KUKA KRL program: f1_Kuka_APT221T02S21.SRC

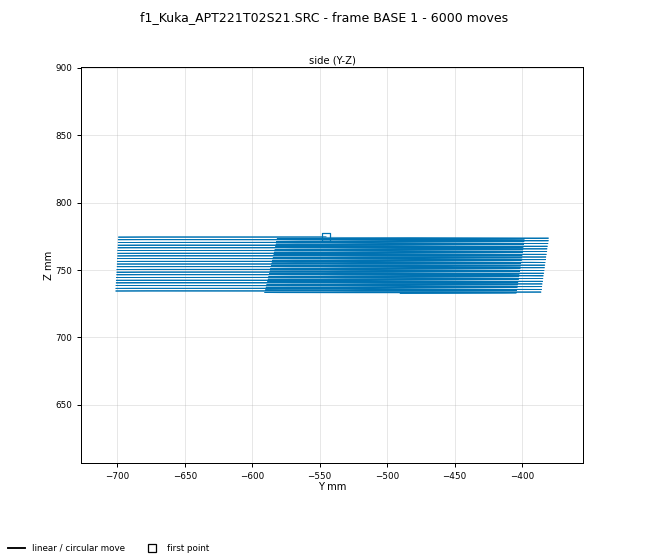
[picture p0: tool path of f1_Kuka_APT221T02S21.SRC in frame BASE 1, 6000 of 6001 moves have a stored position in this frame; points joined in program order, loops and branches not executed]
&ACCESS RVP
&REL 2
&PARAM TEMPLATE = C:\KRC\Roboter\Template\vorgabe
&PARAM EDITMASK = *
DEF f1_Kuka_APT221T02S21()


;FOLD INI;%{PE}%V3.2.0,%MKUKATPBASIS,%CINIT,%VCOMMON,%P
  ;FOLD BAS INI;%{E}%V3.2.0,%MKUKATPBASIS,%CINIT,%VINIT,%P
    GLOBAL INTERRUPT DECL 3 WHEN $STOPMESS==TRUE DO IR_STOPM ( )
    INTERRUPT ON 3
    BAS (#INITMOV,0 )
  ;ENDFOLD (BAS INI)
  ;FOLD USER INI;%{E}%V3.2.0,%MKUKATPUSER,%CINIT,%VINIT,%P
    ;Make your modifications here
  ;ENDFOLD (USER INI)
;ENDFOLD (INI)


;*** Make Null PTP Move
  PTP $pos_act

;*** Auto Load The Correct TOOL Data
  $tool=tool_data[2]

;*** Auto Load The Correct BASE Data
  $base=base_data[1]

  $ADVANCE = 5

;*** Restate Last Velocity
MMPM(30000.0)
SetRPM(8000)
LIN {X 0.178,Y -545.283,Z 774.689,A 0.000,B 0.000,C 90.000,E1 340.007} C_DIS
LIN {X 0.081,Y -552.448,Z 774.686,A 0.000,B 0.000,C 90.000,E1 339.464} C_DIS
LIN {X -0.341,Y -557.944,Z 774.683,A 0.000,B 0.000,C 90.000,E1 339.028} C_DIS
LIN {X 0.055,Y -564.478,Z 774.680,A 0.000,B 0.000,C 90.000,E1 338.358} C_DIS
LIN {X -0.146,Y -569.481,Z 774.677,A 0.000,B 0.000,C 90.000,E1 337.847} C_DIS
LIN {X -0.245,Y -575.503,Z 774.673,A 0.000,B 0.000,C 90.000,E1 337.177} C_DIS
LIN {X -0.071,Y -580.921,Z 774.669,A 0.000,B 0.000,C 90.000,E1 336.485} C_DIS
LIN {X 0.036,Y -588.085,Z 774.664,A 0.000,B 0.000,C 90.000,E1 335.537} C_DIS
LIN {X 0.195,Y -594.819,Z 774.659,A 0.000,B 0.000,C 90.000,E1 334.588} C_DIS
LIN {X -0.171,Y -602.961,Z 774.652,A 0.000,B 0.000,C 90.000,E1 333.435} C_DIS
LIN {X 0.164,Y -608.816,Z 774.647,A 0.000,B 0.000,C 90.000,E1 332.487} C_DIS
LIN {X 0.288,Y -616.060,Z 774.641,A 0.000,B 0.000,C 90.000,E1 331.307} C_DIS
LIN {X -0.314,Y -621.361,Z 774.636,A 0.000,B 0.000,C 90.000,E1 330.461} C_DIS
LIN {X -0.012,Y -626.573,Z 774.631,A 0.000,B 0.000,C 90.000,E1 329.537} C_DIS
LIN {X -0.196,Y -630.736,Z 774.627,A 0.000,B 0.000,C 90.000,E1 328.791} C_DIS
LIN {X 0.216,Y -635.263,Z 774.622,A 0.000,B 0.000,C 90.000,E1 327.867} C_DIS
LIN {X 0.137,Y -639.594,Z 774.617,A 0.000,B 0.000,C 90.000,E1 326.993} C_DIS
LIN {X -0.032,Y -644.812,Z 774.610,A 0.000,B 0.000,C 90.000,E1 325.881} C_DIS
LIN {X 0.321,Y -648.073,Z 774.606,A 0.000,B 0.000,C 90.000,E1 325.102} C_DIS
LIN {X 0.248,Y -652.167,Z 774.601,A 0.000,B 0.000,C 90.000,E1 324.116} C_DIS
LIN {X -0.231,Y -655.030,Z 774.597,A 0.000,B 0.000,C 90.000,E1 323.417} C_DIS
LIN {X -0.278,Y -659.576,Z 774.590,A 0.000,B 0.000,C 90.000,E1 322.190} C_DIS
LIN {X -0.255,Y -663.771,Z 774.583,A 0.000,B 0.000,C 90.000,E1 320.964} C_DIS
LIN {X -0.261,Y -667.644,Z 774.576,A 0.000,B 0.000,C 90.000,E1 319.747} C_DIS
LIN {X -0.199,Y -670.626,Z 774.571,A 0.000,B 0.000,C 90.000,E1 318.771} C_DIS
LIN {X -0.088,Y -674.036,Z 774.564,A 0.000,B 0.000,C 90.000,E1 317.553} C_DIS
LIN {X -0.395,Y -677.421,Z 774.556,A 0.000,B 0.000,C 90.000,E1 316.134} C_DIS
LIN {X -0.247,Y -679.532,Z 774.551,A 0.000,B 0.000,C 90.000,E1 315.162} C_DIS
LIN {X -0.071,Y -681.410,Z 774.546,A 0.000,B 0.000,C 90.000,E1 314.190} C_DIS
LIN {X -0.183,Y -684.457,Z 774.536,A 0.000,B 0.000,C 90.000,E1 312.528} C_DIS
LIN {X 0.094,Y -685.958,Z 774.531,A 0.000,B 0.000,C 90.000,E1 311.553} C_DIS
LIN {X -0.123,Y -687.339,Z 774.526,A 0.000,B 0.000,C 90.000,E1 310.620} C_DIS
LIN {X -0.184,Y -688.796,Z 774.519,A 0.000,B 0.000,C 90.000,E1 309.439} C_DIS
LIN {X -0.219,Y -690.150,Z 774.513,A 0.000,B 0.000,C 90.000,E1 308.257} C_DIS
LIN {X -0.241,Y -691.320,Z 774.506,A 0.000,B 0.000,C 90.000,E1 307.076} C_DIS
LIN {X -0.065,Y -692.595,Z 774.498,A 0.000,B 0.000,C 90.000,E1 305.644} C_DIS
LIN {X 0.083,Y -693.517,Z 774.492,A 0.000,B 0.000,C 90.000,E1 304.452} C_DIS
LIN {X -0.263,Y -694.752,Z 774.482,A 0.000,B 0.000,C 90.000,E1 302.832} C_DIS
LIN {X 0.389,Y -696.099,Z 774.473,A 0.000,B 0.000,C 90.000,E1 301.131} C_DIS
LIN {X -0.157,Y -696.863,Z 774.467,A 0.000,B 0.000,C 90.000,E1 300.001} C_DIS
LIN {X 0.174,Y -697.436,Z 774.459,A 0.000,B 0.000,C 90.000,E1 298.565} C_DIS
LIN {X 0.106,Y -698.271,Z 774.448,A 0.000,B 0.000,C 90.000,E1 296.693} C_DIS
LIN {X 0.045,Y -699.384,Z 774.438,A 0.000,B 0.000,C 90.000,E1 294.823} C_DIS
LIN {X 0.287,Y -699.299,Z 774.435,A 0.000,B 0.000,C 90.000,E1 294.335} C_DIS
LIN {X -0.084,Y -699.187,Z 774.434,A 0.000,B 0.000,C 90.000,E1 294.131} C_DIS
LIN {X 0.162,Y -697.937,Z 774.431,A 0.000,B 0.000,C 90.000,E1 293.643} C_DIS
LIN {X 0.423,Y -697.170,Z 774.430,A 0.000,B 0.000,C 90.000,E1 293.387} C_DIS
LIN {X -0.363,Y -696.496,Z 774.430,A 0.000,B 0.000,C 90.000,E1 293.334} C_DIS
LIN {X -0.234,Y -695.484,Z 774.429,A 0.000,B 0.000,C 90.000,E1 293.206} C_DIS
LIN {X 0.073,Y -690.561,Z 774.426,A 0.000,B 0.000,C 90.000,E1 292.717} C_DIS
LIN {X 0.260,Y -688.711,Z 774.426,A 0.000,B 0.000,C 90.000,E1 292.589} C_DIS
LIN {X -0.357,Y -684.254,Z 774.425,A 0.000,B 0.000,C 90.000,E1 292.461} C_DIS
LIN {X -0.332,Y -680.303,Z 774.424,A 0.000,B 0.000,C 90.000,E1 292.333} C_DIS
LIN {X -0.035,Y -674.173,Z 774.423,A 0.000,B 0.000,C 90.000,E1 292.153} C_DIS
LIN {X -0.204,Y -664.948,Z 774.422,A 0.000,B 0.000,C 90.000,E1 292.025} C_DIS
LIN {X 0.151,Y -654.378,Z 774.422,A 0.000,B 0.000,C 90.000,E1 291.844} C_DIS
LIN {X 0.228,Y -644.131,Z 774.421,A 0.000,B 0.000,C 90.000,E1 291.663} C_DIS
LIN {X -0.242,Y -627.380,Z 774.419,A 0.000,B 0.000,C 90.000,E1 291.354} C_DIS
LIN {X -0.025,Y -610.054,Z 774.416,A 0.000,B 0.000,C 90.000,E1 290.918} C_DIS
LIN {X 0.062,Y -589.210,Z 774.413,A 0.000,B 0.000,C 90.000,E1 290.355} C_DIS
LIN {X -0.059,Y -566.654,Z 774.409,A 0.000,B 0.000,C 90.000,E1 289.685} C_DIS
LIN {X 0.034,Y -560.006,Z 774.408,A 0.000,B 0.000,C 90.000,E1 289.396} C_DIS
LIN {X -0.146,Y -558.225,Z 774.407,A 0.000,B 0.000,C 90.000,E1 289.268} C_DIS
LIN {X 0.119,Y -557.105,Z 774.406,A 0.000,B 0.000,C 90.000,E1 289.141} C_DIS
LIN {X 0.082,Y -557.068,Z 774.406,A 0.000,B 0.000,C 90.000,E1 289.141} C_DIS
LIN {X 0.163,Y -555.965,Z 774.405,A 0.000,B 0.000,C 90.000,E1 288.852} C_DIS
LIN {X 0.333,Y -555.320,Z 774.403,A 0.000,B 0.000,C 90.000,E1 288.417} C_DIS
LIN {X -0.217,Y -554.804,Z 774.398,A 0.000,B 0.000,C 90.000,E1 287.638} C_DIS
LIN {X -0.240,Y -554.409,Z 774.393,A 0.000,B 0.000,C 90.000,E1 286.804} C_DIS
LIN {X 0.088,Y -553.379,Z 774.381,A 0.000,B 0.000,C 90.000,E1 284.537} C_DIS
LIN {X 0.284,Y -552.877,Z 774.373,A 0.000,B 0.000,C 90.000,E1 283.119} C_DIS
LIN {X -0.073,Y -552.310,Z 774.364,A 0.000,B 0.000,C 90.000,E1 281.478} C_DIS
LIN {X 0.115,Y -551.685,Z 774.353,A 0.000,B 0.000,C 90.000,E1 279.500} C_DIS
LIN {X 0.205,Y -551.129,Z 774.342,A 0.000,B 0.000,C 90.000,E1 277.530} C_DIS
LIN {X -0.087,Y -550.812,Z 774.337,A 0.000,B 0.000,C 90.000,E1 276.720} C_DIS
LIN {X 0.206,Y -550.219,Z 774.331,A 0.000,B 0.000,C 90.000,E1 275.568} C_DIS
LIN {X 0.119,Y -548.869,Z 774.320,A 0.000,B 0.000,C 90.000,E1 273.612} C_DIS
LIN {X -0.111,Y -547.883,Z 774.311,A 0.000,B 0.000,C 90.000,E1 271.949} C_DIS
LIN {X 0.092,Y -547.188,Z 774.305,A 0.000,B 0.000,C 90.000,E1 270.802} C_DIS
LIN {X -0.187,Y -546.082,Z 774.295,A 0.000,B 0.000,C 90.000,E1 269.141} C_DIS
LIN {X 0.101,Y -544.746,Z 774.284,A 0.000,B 0.000,C 90.000,E1 267.135} C_DIS
LIN {X -0.194,Y -543.673,Z 774.275,A 0.000,B 0.000,C 90.000,E1 265.469} C_DIS
LIN {X 0.008,Y -542.820,Z 774.267,A 0.000,B 0.000,C 90.000,E1 264.033} C_DIS
LIN {X 0.239,Y -541.958,Z 774.261,A 0.000,B 0.000,C 90.000,E1 262.875} C_DIS
LIN {X 0.134,Y -539.840,Z 774.246,A 0.000,B 0.000,C 90.000,E1 260.330} C_DIS
LIN {X 0.029,Y -538.329,Z 774.237,A 0.000,B 0.000,C 90.000,E1 258.634} C_DIS
LIN {X -0.164,Y -537.057,Z 774.229,A 0.000,B 0.000,C 90.000,E1 257.229} C_DIS
LIN {X 0.074,Y -536.003,Z 774.223,A 0.000,B 0.000,C 90.000,E1 256.061} C_DIS
LIN {X 0.176,Y -533.831,Z 774.212,A 0.000,B 0.000,C 90.000,E1 254.047} C_DIS
LIN {X 0.017,Y -531.551,Z 774.200,A 0.000,B 0.000,C 90.000,E1 252.054} C_DIS
LIN {X -0.069,Y -530.230,Z 774.194,A 0.000,B 0.000,C 90.000,E1 250.913} C_DIS
LIN {X 0.174,Y -527.788,Z 774.184,A 0.000,B 0.000,C 90.000,E1 249.156} C_DIS
LIN {X 0.077,Y -525.719,Z 774.176,A 0.000,B 0.000,C 90.000,E1 247.720} C_DIS
LIN {X 0.278,Y -522.634,Z 774.165,A 0.000,B 0.000,C 90.000,E1 245.665} C_DIS
LIN {X -0.010,Y -519.775,Z 774.155,A 0.000,B 0.000,C 90.000,E1 243.948} C_DIS
LIN {X -0.028,Y -517.319,Z 774.147,A 0.000,B 0.000,C 90.000,E1 242.487} C_DIS
LIN {X 0.118,Y -515.723,Z 774.142,A 0.000,B 0.000,C 90.000,E1 241.591} C_DIS
LIN {X 0.142,Y -513.476,Z 774.136,A 0.000,B 0.000,C 90.000,E1 240.411} C_DIS
LIN {X 0.032,Y -510.654,Z 774.128,A 0.000,B 0.000,C 90.000,E1 238.948} C_DIS
LIN {X -0.192,Y -508.290,Z 774.121,A 0.000,B 0.000,C 90.000,E1 237.788} C_DIS
LIN {X -0.063,Y -506.493,Z 774.116,A 0.000,B 0.000,C 90.000,E1 236.882} C_DIS
LIN {X -0.231,Y -504.589,Z 774.111,A 0.000,B 0.000,C 90.000,E1 236.008} C_DIS
LIN {X 0.157,Y -501.831,Z 774.104,A 0.000,B 0.000,C 90.000,E1 234.769} C_DIS
LIN {X -0.194,Y -499.657,Z 774.099,A 0.000,B 0.000,C 90.000,E1 233.909} C_DIS
LIN {X -0.127,Y -495.856,Z 774.091,A 0.000,B 0.000,C 90.000,E1 232.396} C_DIS
LIN {X 0.028,Y -491.385,Z 774.081,A 0.000,B 0.000,C 90.000,E1 230.561} C_DIS
LIN {X 0.038,Y -485.694,Z 774.067,A 0.000,B 0.000,C 90.000,E1 228.119} C_DIS
LIN {X 0.124,Y -480.447,Z 774.054,A 0.000,B 0.000,C 90.000,E1 225.648} C_DIS
LIN {X 0.057,Y -477.077,Z 774.045,A 0.000,B 0.000,C 90.000,E1 224.109} C_DIS
LIN {X 0.267,Y -473.705,Z 774.036,A 0.000,B 0.000,C 90.000,E1 222.528} C_DIS
LIN {X -0.295,Y -468.229,Z 774.023,A 0.000,B 0.000,C 90.000,E1 220.092} C_DIS
LIN {X -0.103,Y -464.205,Z 774.012,A 0.000,B 0.000,C 90.000,E1 218.177} C_DIS
LIN {X -0.037,Y -460.932,Z 774.003,A 0.000,B 0.000,C 90.000,E1 216.583} C_DIS
LIN {X -0.050,Y -458.321,Z 773.996,A 0.000,B 0.000,C 90.000,E1 215.311} C_DIS
LIN {X -0.081,Y -453.083,Z 773.982,A 0.000,B 0.000,C 90.000,E1 212.752} C_DIS
LIN {X -0.091,Y -450.570,Z 773.975,A 0.000,B 0.000,C 90.000,E1 211.465} C_DIS
LIN {X -0.149,Y -446.255,Z 773.962,A 0.000,B 0.000,C 90.000,E1 209.205} C_DIS
LIN {X -0.207,Y -442.547,Z 773.951,A 0.000,B 0.000,C 90.000,E1 207.257} C_DIS
LIN {X 0.004,Y -439.406,Z 773.942,A 0.000,B 0.000,C 90.000,E1 205.591} C_DIS
LIN {X -0.040,Y -436.335,Z 773.933,A 0.000,B 0.000,C 90.000,E1 203.951} C_DIS
LIN {X 0.084,Y -433.208,Z 773.924,A 0.000,B 0.000,C 90.000,E1 202.280} C_DIS
LIN {X -0.041,Y -429.452,Z 773.913,A 0.000,B 0.000,C 90.000,E1 200.301} C_DIS
LIN {X -0.149,Y -425.598,Z 773.902,A 0.000,B 0.000,C 90.000,E1 198.308} C_DIS
LIN {X 0.217,Y -423.052,Z 773.894,A 0.000,B 0.000,C 90.000,E1 196.913} C_DIS
LIN {X -0.125,Y -418.385,Z 773.881,A 0.000,B 0.000,C 90.000,E1 194.592} C_DIS
LIN {X 0.019,Y -413.939,Z 773.868,A 0.000,B 0.000,C 90.000,E1 192.187} C_DIS
LIN {X -0.036,Y -409.702,Z 773.854,A 0.000,B 0.000,C 90.000,E1 189.792} C_DIS
LIN {X 0.100,Y -406.128,Z 773.843,A 0.000,B 0.000,C 90.000,E1 187.701} C_DIS
LIN {X 0.081,Y -403.234,Z 773.833,A 0.000,B 0.000,C 90.000,E1 185.967} C_DIS
LIN {X -0.194,Y -398.831,Z 773.818,A 0.000,B 0.000,C 90.000,E1 183.212} C_DIS
LIN {X 0.044,Y -394.221,Z 773.798,A 0.000,B 0.000,C 90.000,E1 179.656} C_DIS
LIN {X 0.094,Y -390.347,Z 773.778,A 0.000,B 0.000,C 90.000,E1 176.102} C_DIS
LIN {X 0.111,Y -388.733,Z 773.769,A 0.000,B 0.000,C 90.000,E1 174.318} C_DIS
LIN {X -0.103,Y -386.282,Z 773.753,A 0.000,B 0.000,C 90.000,E1 171.489} C_DIS
LIN {X -0.140,Y -384.498,Z 773.739,A 0.000,B 0.000,C 90.000,E1 168.982} C_DIS
LIN {X -0.070,Y -383.343,Z 773.729,A 0.000,B 0.000,C 90.000,E1 167.173} C_DIS
LIN {X 0.060,Y -382.116,Z 773.715,A 0.000,B 0.000,C 90.000,E1 164.629} C_DIS
LIN {X -0.117,Y -381.087,Z 773.701,A 0.000,B 0.000,C 90.000,E1 162.127} C_DIS
LIN {X 0.028,Y -380.380,Z 773.687,A 0.000,B 0.000,C 90.000,E1 159.571} C_DIS
LIN {X 0.136,Y -380.243,Z 773.660,A 0.000,B 0.000,C 90.000,E1 154.845} C_DIS
LIN {X 0.216,Y -382.155,Z 773.634,A 0.000,B 0.000,C 90.000,E1 150.127} C_DIS
LIN {X -0.174,Y -384.714,Z 773.620,A 0.000,B 0.000,C 90.000,E1 147.661} C_DIS
LIN {X 0.085,Y -387.767,Z 773.608,A 0.000,B 0.000,C 90.000,E1 145.468} C_DIS
LIN {X 0.035,Y -389.915,Z 773.602,A 0.000,B 0.000,C 90.000,E1 144.402} C_DIS
LIN {X 0.013,Y -392.530,Z 773.596,A 0.000,B 0.000,C 90.000,E1 143.336} C_DIS
LIN {X -0.064,Y -394.697,Z 773.592,A 0.000,B 0.000,C 90.000,E1 142.637} C_DIS
LIN {X 0.022,Y -395.970,Z 773.590,A 0.000,B 0.000,C 90.000,E1 142.271} C_DIS
LIN {X 0.034,Y -398.582,Z 773.587,A 0.000,B 0.000,C 90.000,E1 141.662} C_DIS
LIN {X -0.058,Y -401.787,Z 773.584,A 0.000,B 0.000,C 90.000,E1 141.090} C_DIS
LIN {X 0.210,Y -405.826,Z 773.580,A 0.000,B 0.000,C 90.000,E1 140.436} C_DIS
LIN {X 0.202,Y -410.581,Z 773.577,A 0.000,B 0.000,C 90.000,E1 139.828} C_DIS
LIN {X 0.147,Y -421.432,Z 773.570,A 0.000,B 0.000,C 90.000,E1 138.609} C_DIS
LIN {X -0.120,Y -438.562,Z 773.560,A 0.000,B 0.000,C 90.000,E1 136.824} C_DIS
LIN {X 0.061,Y -447.060,Z 773.555,A 0.000,B 0.000,C 90.000,E1 135.891} C_DIS
LIN {X -0.217,Y -452.568,Z 773.552,A 0.000,B 0.000,C 90.000,E1 135.324} C_DIS
LIN {X 0.068,Y -458.023,Z 773.548,A 0.000,B 0.000,C 90.000,E1 134.676} C_DIS
LIN {X 0.224,Y -462.048,Z 773.546,A 0.000,B 0.000,C 90.000,E1 134.190} C_DIS
LIN {X -0.056,Y -470.928,Z 773.540,A 0.000,B 0.000,C 90.000,E1 133.137} C_DIS
LIN {X -0.058,Y -479.685,Z 773.534,A 0.000,B 0.000,C 90.000,E1 132.043} C_DIS
LIN {X 0.030,Y -486.658,Z 773.528,A 0.000,B 0.000,C 90.000,E1 131.105} C_DIS
LIN {X 0.078,Y -492.129,Z 773.524,A 0.000,B 0.000,C 90.000,E1 130.334} C_DIS
LIN {X 0.127,Y -500.272,Z 773.517,A 0.000,B 0.000,C 90.000,E1 129.116} C_DIS
LIN {X -0.133,Y -506.692,Z 773.512,A 0.000,B 0.000,C 90.000,E1 128.096} C_DIS
LIN {X 0.291,Y -511.891,Z 773.507,A 0.000,B 0.000,C 90.000,E1 127.156} C_DIS
LIN {X -0.012,Y -518.359,Z 773.500,A 0.000,B 0.000,C 90.000,E1 126.011} C_DIS
LIN {X -0.120,Y -522.871,Z 773.495,A 0.000,B 0.000,C 90.000,E1 125.152} C_DIS
LIN {X 0.221,Y -525.752,Z 773.492,A 0.000,B 0.000,C 90.000,E1 124.532} C_DIS
LIN {X 0.017,Y -527.695,Z 773.490,A 0.000,B 0.000,C 90.000,E1 124.119} C_DIS
LIN {X -0.336,Y -530.307,Z 773.486,A 0.000,B 0.000,C 90.000,E1 123.579} C_DIS
LIN {X -0.249,Y -535.183,Z 773.480,A 0.000,B 0.000,C 90.000,E1 122.418} C_DIS
LIN {X -0.099,Y -538.587,Z 773.475,A 0.000,B 0.000,C 90.000,E1 121.544} C_DIS
LIN {X 0.089,Y -541.752,Z 773.470,A 0.000,B 0.000,C 90.000,E1 120.669} C_DIS
LIN {X 0.309,Y -544.729,Z 773.466,A 0.000,B 0.000,C 90.000,E1 119.795} C_DIS
LIN {X 0.045,Y -548.454,Z 773.459,A 0.000,B 0.000,C 90.000,E1 118.693} C_DIS
LIN {X -0.165,Y -551.979,Z 773.453,A 0.000,B 0.000,C 90.000,E1 117.590} C_DIS
LIN {X 0.120,Y -553.550,Z 773.450,A 0.000,B 0.000,C 90.000,E1 117.001} C_DIS
LIN {X 0.168,Y -555.023,Z 773.447,A 0.000,B 0.000,C 90.000,E1 116.437} C_DIS
LIN {X 0.041,Y -557.322,Z 773.441,A 0.000,B 0.000,C 90.000,E1 115.335} C_DIS
LIN {X 0.119,Y -558.335,Z 773.438,A 0.000,B 0.000,C 90.000,E1 114.771} C_DIS
LIN {X -0.002,Y -559.571,Z 773.433,A 0.000,B 0.000,C 90.000,E1 113.951} C_DIS
LIN {X -0.120,Y -562.016,Z 773.422,A 0.000,B 0.000,C 90.000,E1 112.025} C_DIS
LIN {X -0.101,Y -563.264,Z 773.416,A 0.000,B 0.000,C 90.000,E1 110.918} C_DIS
LIN {X 0.068,Y -564.689,Z 773.409,A 0.000,B 0.000,C 90.000,E1 109.523} C_DIS
LIN {X 0.118,Y -565.726,Z 773.402,A 0.000,B 0.000,C 90.000,E1 108.417} C_DIS
LIN {X -0.231,Y -567.099,Z 773.393,A 0.000,B 0.000,C 90.000,E1 106.804} C_DIS
LIN {X -0.001,Y -568.475,Z 773.384,A 0.000,B 0.000,C 90.000,E1 105.134} C_DIS
LIN {X -0.125,Y -570.072,Z 773.373,A 0.000,B 0.000,C 90.000,E1 103.231} C_DIS
LIN {X -0.118,Y -571.532,Z 773.364,A 0.000,B 0.000,C 90.000,E1 101.591} C_DIS
LIN {X -0.189,Y -573.046,Z 773.355,A 0.000,B 0.000,C 90.000,E1 99.962} C_DIS
LIN {X 0.140,Y -574.192,Z 773.348,A 0.000,B 0.000,C 90.000,E1 98.568} C_DIS
LIN {X -0.164,Y -575.283,Z 773.340,A 0.000,B 0.000,C 90.000,E1 97.239} C_DIS
LIN {X 0.121,Y -576.219,Z 773.333,A 0.000,B 0.000,C 90.000,E1 95.853} C_DIS
LIN {X -0.212,Y -577.072,Z 773.325,A 0.000,B 0.000,C 90.000,E1 94.531} C_DIS
LIN {X 0.010,Y -577.964,Z 773.318,A 0.000,B 0.000,C 90.000,E1 93.154} C_DIS
LIN {X -0.145,Y -578.806,Z 773.309,A 0.000,B 0.000,C 90.000,E1 91.547} C_DIS
LIN {X 0.257,Y -579.567,Z 773.300,A 0.000,B 0.000,C 90.000,E1 89.885} C_DIS
LIN {X -0.237,Y -580.006,Z 773.294,A 0.000,B 0.000,C 90.000,E1 88.854} C_DIS
LIN {X 0.201,Y -580.539,Z 773.285,A 0.000,B 0.000,C 90.000,E1 87.192} C_DIS
LIN {X 0.102,Y -580.981,Z 773.276,A 0.000,B 0.000,C 90.000,E1 85.584} C_DIS
LIN {X 0.068,Y -581.295,Z 773.267,A 0.000,B 0.000,C 90.000,E1 83.970} C_DIS
LIN {X 0.041,Y -581.498,Z 773.258,A 0.000,B 0.000,C 90.000,E1 82.356} C_DIS
LIN {X 0.086,Y -581.606,Z 773.249,A 0.000,B 0.000,C 90.000,E1 80.735} C_DIS
LIN {X -0.006,Y -581.651,Z 773.241,A 0.000,B 0.000,C 90.000,E1 79.398} C_DIS
LIN {X -0.218,Y -581.605,Z 773.235,A 0.000,B 0.000,C 90.000,E1 78.342} C_DIS
LIN {X 0.036,Y -581.372,Z 773.226,A 0.000,B 0.000,C 90.000,E1 76.700} C_DIS
LIN {X 0.042,Y -580.986,Z 773.219,A 0.000,B 0.000,C 90.000,E1 75.353} C_DIS
LIN {X -0.223,Y -580.524,Z 773.211,A 0.000,B 0.000,C 90.000,E1 74.031} C_DIS
LIN {X -0.098,Y -580.048,Z 773.204,A 0.000,B 0.000,C 90.000,E1 72.670} C_DIS
LIN {X 0.009,Y -579.324,Z 773.195,A 0.000,B 0.000,C 90.000,E1 71.040} C_DIS
LIN {X 0.295,Y -578.426,Z 773.186,A 0.000,B 0.000,C 90.000,E1 69.390} C_DIS
LIN {X 0.175,Y -577.552,Z 773.178,A 0.000,B 0.000,C 90.000,E1 68.050} C_DIS
LIN {X 0.095,Y -576.727,Z 773.172,A 0.000,B 0.000,C 90.000,E1 66.975} C_DIS
LIN {X 0.157,Y -575.586,Z 773.165,A 0.000,B 0.000,C 90.000,E1 65.613} C_DIS
LIN {X 0.060,Y -574.514,Z 773.159,A 0.000,B 0.000,C 90.000,E1 64.537} C_DIS
LIN {X -0.052,Y -573.295,Z 773.153,A 0.000,B 0.000,C 90.000,E1 63.461} C_DIS
LIN {X 0.236,Y -572.274,Z 773.148,A 0.000,B 0.000,C 90.000,E1 62.615} C_DIS
LIN {X -0.153,Y -570.637,Z 773.142,A 0.000,B 0.000,C 90.000,E1 61.563} C_DIS
LIN {X 0.114,Y -569.305,Z 773.137,A 0.000,B 0.000,C 90.000,E1 60.717} C_DIS
LIN {X 0.179,Y -567.276,Z 773.131,A 0.000,B 0.000,C 90.000,E1 59.616} C_DIS
LIN {X 0.009,Y -564.956,Z 773.125,A 0.000,B 0.000,C 90.000,E1 58.535} C_DIS
LIN {X 0.014,Y -562.945,Z 773.121,A 0.000,B 0.000,C 90.000,E1 57.709} C_DIS
LIN {X -0.302,Y -560.777,Z 773.116,A 0.000,B 0.000,C 90.000,E1 56.914} C_DIS
LIN {X -0.338,Y -558.377,Z 773.111,A 0.000,B 0.000,C 90.000,E1 56.087} C_DIS
LIN {X -0.083,Y -555.765,Z 773.107,A 0.000,B 0.000,C 90.000,E1 55.229} C_DIS
LIN {X -0.244,Y -553.974,Z 773.104,A 0.000,B 0.000,C 90.000,E1 54.689} C_DIS
LIN {X -0.033,Y -550.883,Z 773.099,A 0.000,B 0.000,C 90.000,E1 53.829} C_DIS
LIN {X 0.147,Y -547.370,Z 773.094,A 0.000,B 0.000,C 90.000,E1 52.970} C_DIS
LIN {X 0.098,Y -544.221,Z 773.091,A 0.000,B 0.000,C 90.000,E1 52.271} C_DIS
LIN {X 0.347,Y -540.776,Z 773.087,A 0.000,B 0.000,C 90.000,E1 51.537} C_DIS
LIN {X -0.032,Y -537.828,Z 773.083,A 0.000,B 0.000,C 90.000,E1 51.009} C_DIS
LIN {X -0.013,Y -534.607,Z 773.080,A 0.000,B 0.000,C 90.000,E1 50.436} C_DIS
LIN {X 0.321,Y -531.003,Z 773.077,A 0.000,B 0.000,C 90.000,E1 49.828} C_DIS
LIN {X -0.119,Y -527.038,Z 773.074,A 0.000,B 0.000,C 90.000,E1 49.299} C_DIS
LIN {X 0.157,Y -522.515,Z 773.071,A 0.000,B 0.000,C 90.000,E1 48.690} C_DIS
LIN {X 0.049,Y -517.571,Z 773.067,A 0.000,B 0.000,C 90.000,E1 48.119} C_DIS
LIN {X -0.118,Y -513.694,Z 773.065,A 0.000,B 0.000,C 90.000,E1 47.715} C_DIS
LIN {X 0.267,Y -508.407,Z 773.062,A 0.000,B 0.000,C 90.000,E1 47.148} C_DIS
LIN {X 0.013,Y -502.833,Z 773.059,A 0.000,B 0.000,C 90.000,E1 46.662} C_DIS
LIN {X 0.150,Y -496.641,Z 773.056,A 0.000,B 0.000,C 90.000,E1 46.134} C_DIS
LIN {X -0.169,Y -488.987,Z 773.053,A 0.000,B 0.000,C 90.000,E1 45.567} C_DIS
LIN {X 0.007,Y -482.603,Z 773.050,A 0.000,B 0.000,C 90.000,E1 45.081} C_DIS
LIN {X 0.121,Y -474.562,Z 773.047,A 0.000,B 0.000,C 90.000,E1 44.514} C_DIS
LIN {X -0.115,Y -463.153,Z 773.043,A 0.000,B 0.000,C 90.000,E1 43.785} C_DIS
LIN {X -0.192,Y -445.398,Z 773.037,A 0.000,B 0.000,C 90.000,E1 42.609} C_DIS
LIN {X 0.128,Y -421.634,Z 773.027,A 0.000,B 0.000,C 90.000,E1 40.862} C_DIS
LIN {X -0.201,Y -412.507,Z 773.023,A 0.000,B 0.000,C 90.000,E1 40.172} C_DIS
LIN {X -0.109,Y -407.890,Z 773.021,A 0.000,B 0.000,C 90.000,E1 39.725} C_DIS
LIN {X -0.141,Y -407.878,Z 773.021,A 0.000,B 0.000,C 90.000,E1 39.725} C_DIS
LIN {X 0.119,Y -405.989,Z 773.014,A 0.000,B 0.000,C 90.000,E1 38.543} C_DIS
LIN {X -0.095,Y -398.283,Z 772.993,A 0.000,B 0.000,C 90.000,E1 34.739} C_DIS
LIN {X 0.121,Y -398.143,Z 772.992,A 0.000,B 0.000,C 90.000,E1 34.532} C_DIS
LIN {X 0.133,Y -398.801,Z 772.975,A 0.000,B 0.000,C 90.000,E1 31.544} C_DIS
LIN {X -0.032,Y -400.127,Z 772.958,A 0.000,B 0.000,C 90.000,E1 28.409} C_DIS
LIN {X 0.089,Y -401.759,Z 772.942,A 0.000,B 0.000,C 90.000,E1 25.591} C_DIS
LIN {X 0.012,Y -403.955,Z 772.925,A 0.000,B 0.000,C 90.000,E1 22.461} C_DIS
LIN {X -0.080,Y -407.648,Z 772.904,A 0.000,B 0.000,C 90.000,E1 18.652} C_DIS
LIN {X -0.004,Y -412.203,Z 772.884,A 0.000,B 0.000,C 90.000,E1 15.190} C_DIS
LIN {X 0.127,Y -415.859,Z 772.871,A 0.000,B 0.000,C 90.000,E1 12.771} C_DIS
LIN {X 0.067,Y -418.662,Z 772.862,A 0.000,B 0.000,C 90.000,E1 11.074} C_DIS
LIN {X 0.128,Y -422.097,Z 772.850,A 0.000,B 0.000,C 90.000,E1 9.029} C_DIS
LIN {X 0.041,Y -425.031,Z 772.841,A 0.000,B 0.000,C 90.000,E1 7.352} C_DIS
LIN {X 0.207,Y -429.677,Z 772.826,A 0.000,B 0.000,C 90.000,E1 4.645} C_DIS
LIN {X 0.001,Y -434.656,Z 772.811,A 0.000,B 0.000,C 90.000,E1 2.007} C_DIS
LIN {X 0.059,Y -437.834,Z 772.802,A 0.000,B 0.000,C 90.000,E1 0.344} C_DIS
LIN {X 0.063,Y -441.000,Z 772.793,A 0.000,B 0.000,C 90.000,E1 358.797} C_DIS
LIN {X 0.085,Y -445.908,Z 772.781,A 0.000,B 0.000,C 90.000,E1 356.502} C_DIS
LIN {X 0.089,Y -450.449,Z 772.770,A 0.000,B 0.000,C 90.000,E1 354.552} C_DIS
LIN {X 0.127,Y -454.236,Z 772.761,A 0.000,B 0.000,C 90.000,E1 352.932} C_DIS
LIN {X 0.184,Y -457.937,Z 772.752,A 0.000,B 0.000,C 90.000,E1 351.319} C_DIS
LIN {X -0.032,Y -460.111,Z 772.747,A 0.000,B 0.000,C 90.000,E1 350.387} C_DIS
LIN {X 0.026,Y -462.873,Z 772.740,A 0.000,B 0.000,C 90.000,E1 349.106} C_DIS
LIN {X 0.091,Y -467.764,Z 772.727,A 0.000,B 0.000,C 90.000,E1 346.881} C_DIS
LIN {X -0.181,Y -469.533,Z 772.724,A 0.000,B 0.000,C 90.000,E1 346.284} C_DIS
LIN {X -0.011,Y -471.921,Z 772.720,A 0.000,B 0.000,C 90.000,E1 345.644} C_DIS
LIN {X -0.070,Y -473.509,Z 772.719,A 0.000,B 0.000,C 90.000,E1 345.338} C_DIS
LIN {X -0.038,Y -476.510,Z 772.716,A 0.000,B 0.000,C 90.000,E1 344.866} C_DIS
LIN {X -0.215,Y -480.729,Z 772.713,A 0.000,B 0.000,C 90.000,E1 344.393} C_DIS
LIN {X -0.146,Y -486.361,Z 772.710,A 0.000,B 0.000,C 90.000,E1 343.850} C_DIS
LIN {X 0.176,Y -494.236,Z 772.707,A 0.000,B 0.000,C 90.000,E1 343.196} C_DIS
LIN {X 0.007,Y -514.551,Z 772.699,A 0.000,B 0.000,C 90.000,E1 341.819} C_DIS
LIN {X 0.128,Y -533.439,Z 772.692,A 0.000,B 0.000,C 90.000,E1 340.604} C_DIS
LIN {X 0.019,Y -542.864,Z 772.689,A 0.000,B 0.000,C 90.000,E1 340.007} C_DIS
LIN {X 0.231,Y -550.201,Z 772.686,A 0.000,B 0.000,C 90.000,E1 339.444} C_DIS
LIN {X -0.083,Y -554.400,Z 772.684,A 0.000,B 0.000,C 90.000,E1 339.135} C_DIS
LIN {X -0.050,Y -561.128,Z 772.681,A 0.000,B 0.000,C 90.000,E1 338.518} C_DIS
LIN {X -0.070,Y -566.024,Z 772.678,A 0.000,B 0.000,C 90.000,E1 338.028} C_DIS
LIN {X -0.103,Y -572.205,Z 772.674,A 0.000,B 0.000,C 90.000,E1 337.358} C_DIS
LIN {X 0.088,Y -576.850,Z 772.671,A 0.000,B 0.000,C 90.000,E1 336.794} C_DIS
LIN {X -0.015,Y -583.288,Z 772.667,A 0.000,B 0.000,C 90.000,E1 335.997} C_DIS
LIN {X 0.079,Y -590.319,Z 772.661,A 0.000,B 0.000,C 90.000,E1 335.049} C_DIS
LIN {X -0.276,Y -596.902,Z 772.656,A 0.000,B 0.000,C 90.000,E1 334.152} C_DIS
LIN {X 0.019,Y -602.396,Z 772.652,A 0.000,B 0.000,C 90.000,E1 333.332} C_DIS
LIN {X 0.107,Y -607.503,Z 772.648,A 0.000,B 0.000,C 90.000,E1 332.538} C_DIS
LIN {X -0.046,Y -613.246,Z 772.642,A 0.000,B 0.000,C 90.000,E1 331.641} C_DIS
LIN {X 0.169,Y -617.971,Z 772.638,A 0.000,B 0.000,C 90.000,E1 330.845} C_DIS
LIN {X -0.100,Y -626.265,Z 772.630,A 0.000,B 0.000,C 90.000,E1 329.459} C_DIS
LIN {X 0.261,Y -631.094,Z 772.625,A 0.000,B 0.000,C 90.000,E1 328.535} C_DIS
LIN {X -0.368,Y -636.996,Z 772.619,A 0.000,B 0.000,C 90.000,E1 327.454} C_DIS
LIN {X -0.037,Y -642.357,Z 772.613,A 0.000,B 0.000,C 90.000,E1 326.294} C_DIS
LIN {X -0.192,Y -646.891,Z 772.607,A 0.000,B 0.000,C 90.000,E1 325.308} C_DIS
LIN {X 0.246,Y -651.051,Z 772.602,A 0.000,B 0.000,C 90.000,E1 324.276} C_DIS
LIN {X 0.141,Y -654.023,Z 772.598,A 0.000,B 0.000,C 90.000,E1 323.543} C_DIS
LIN {X 0.140,Y -657.738,Z 772.592,A 0.000,B 0.000,C 90.000,E1 322.557} C_DIS
LIN {X 0.108,Y -660.360,Z 772.588,A 0.000,B 0.000,C 90.000,E1 321.823} C_DIS
LIN {X -0.343,Y -663.740,Z 772.583,A 0.000,B 0.000,C 90.000,E1 320.884} C_DIS
LIN {X -0.336,Y -666.938,Z 772.577,A 0.000,B 0.000,C 90.000,E1 319.908} C_DIS
LIN {X -0.284,Y -670.675,Z 772.570,A 0.000,B 0.000,C 90.000,E1 318.690} C_DIS
LIN {X -0.171,Y -674.065,Z 772.564,A 0.000,B 0.000,C 90.000,E1 317.472} C_DIS
LIN {X -0.006,Y -677.513,Z 772.556,A 0.000,B 0.000,C 90.000,E1 316.014} C_DIS
LIN {X -0.328,Y -679.664,Z 772.550,A 0.000,B 0.000,C 90.000,E1 315.081} C_DIS
LIN {X -0.150,Y -681.567,Z 772.545,A 0.000,B 0.000,C 90.000,E1 314.109} C_DIS
LIN {X -0.314,Y -684.197,Z 772.537,A 0.000,B 0.000,C 90.000,E1 312.690} C_DIS
LIN {X 0.416,Y -685.790,Z 772.532,A 0.000,B 0.000,C 90.000,E1 311.676} C_DIS
LIN {X -0.256,Y -687.241,Z 772.526,A 0.000,B 0.000,C 90.000,E1 310.782} C_DIS
LIN {X 0.123,Y -688.750,Z 772.520,A 0.000,B 0.000,C 90.000,E1 309.564} C_DIS
LIN {X -0.290,Y -690.371,Z 772.512,A 0.000,B 0.000,C 90.000,E1 308.177} C_DIS
LIN {X 0.241,Y -691.570,Z 772.505,A 0.000,B 0.000,C 90.000,E1 306.950} C_DIS
LIN {X 0.429,Y -692.840,Z 772.498,A 0.000,B 0.000,C 90.000,E1 305.518} C_DIS
LIN {X -0.379,Y -693.754,Z 772.491,A 0.000,B 0.000,C 90.000,E1 304.405} C_DIS
LIN {X -0.333,Y -694.993,Z 772.482,A 0.000,B 0.000,C 90.000,E1 302.752} C_DIS
LIN {X -0.041,Y -696.305,Z 772.473,A 0.000,B 0.000,C 90.000,E1 301.082} C_DIS
LIN {X -0.229,Y -697.063,Z 772.466,A 0.000,B 0.000,C 90.000,E1 299.922} C_DIS
LIN {X 0.099,Y -697.599,Z 772.458,A 0.000,B 0.000,C 90.000,E1 298.487} C_DIS
LIN {X 0.118,Y -698.203,Z 772.451,A 0.000,B 0.000,C 90.000,E1 297.078} C_DIS
LIN {X 0.030,Y -699.381,Z 772.439,A 0.000,B 0.000,C 90.000,E1 294.975} C_DIS
LIN {X -0.335,Y -699.511,Z 772.438,A 0.000,B 0.000,C 90.000,E1 294.771} C_DIS
LIN {X 0.198,Y -699.315,Z 772.435,A 0.000,B 0.000,C 90.000,E1 294.259} C_DIS
LIN {X 0.179,Y -699.078,Z 772.434,A 0.000,B 0.000,C 90.000,E1 294.027} C_DIS
LIN {X 0.068,Y -697.674,Z 772.431,A 0.000,B 0.000,C 90.000,E1 293.567} C_DIS
LIN {X 0.051,Y -696.688,Z 772.430,A 0.000,B 0.000,C 90.000,E1 293.334} C_DIS
LIN {X 0.180,Y -695.782,Z 772.429,A 0.000,B 0.000,C 90.000,E1 293.206} C_DIS
LIN {X -0.309,Y -692.103,Z 772.427,A 0.000,B 0.000,C 90.000,E1 292.898} C_DIS
LIN {X -0.136,Y -690.756,Z 772.427,A 0.000,B 0.000,C 90.000,E1 292.770} C_DIS
LIN {X 0.038,Y -689.103,Z 772.426,A 0.000,B 0.000,C 90.000,E1 292.642} C_DIS
LIN {X -0.137,Y -684.355,Z 772.425,A 0.000,B 0.000,C 90.000,E1 292.461} C_DIS
LIN {X -0.175,Y -680.063,Z 772.424,A 0.000,B 0.000,C 90.000,E1 292.333} C_DIS
LIN {X -0.286,Y -674.745,Z 772.423,A 0.000,B 0.000,C 90.000,E1 292.206} C_DIS
LIN {X 0.230,Y -666.220,Z 772.423,A 0.000,B 0.000,C 90.000,E1 292.025} C_DIS
LIN {X 0.299,Y -657.093,Z 772.422,A 0.000,B 0.000,C 90.000,E1 291.897} C_DIS
LIN {X -0.175,Y -643.701,Z 772.421,A 0.000,B 0.000,C 90.000,E1 291.716} C_DIS
LIN {X -0.085,Y -626.945,Z 772.419,A 0.000,B 0.000,C 90.000,E1 291.354} C_DIS
LIN {X 0.084,Y -609.530,Z 772.416,A 0.000,B 0.000,C 90.000,E1 290.918} C_DIS
LIN {X -0.073,Y -588.716,Z 772.413,A 0.000,B 0.000,C 90.000,E1 290.375} C_DIS
LIN {X 0.031,Y -566.086,Z 772.409,A 0.000,B 0.000,C 90.000,E1 289.685} C_DIS
LIN {X 0.223,Y -559.755,Z 772.408,A 0.000,B 0.000,C 90.000,E1 289.396} C_DIS
LIN {X 0.230,Y -558.790,Z 772.408,A 0.000,B 0.000,C 90.000,E1 289.322} C_DIS
LIN {X -0.284,Y -556.981,Z 772.407,A 0.000,B 0.000,C 90.000,E1 289.214} C_DIS
LIN {X -0.321,Y -556.940,Z 772.407,A 0.000,B 0.000,C 90.000,E1 289.214} C_DIS
LIN {X 0.015,Y -556.042,Z 772.405,A 0.000,B 0.000,C 90.000,E1 288.960} C_DIS
LIN {X -0.096,Y -555.485,Z 772.404,A 0.000,B 0.000,C 90.000,E1 288.671} C_DIS
LIN {X -0.224,Y -554.987,Z 772.401,A 0.000,B 0.000,C 90.000,E1 288.127} C_DIS
LIN {X 0.036,Y -554.516,Z 772.394,A 0.000,B 0.000,C 90.000,E1 286.985} C_DIS
LIN {X -0.044,Y -553.384,Z 772.380,A 0.000,B 0.000,C 90.000,E1 284.481} C_DIS
LIN {X 0.155,Y -552.879,Z 772.373,A 0.000,B 0.000,C 90.000,E1 283.063} C_DIS
LIN {X -0.199,Y -552.321,Z 772.363,A 0.000,B 0.000,C 90.000,E1 281.422} C_DIS
LIN {X -0.008,Y -551.667,Z 772.353,A 0.000,B 0.000,C 90.000,E1 279.443} C_DIS
LIN {X 0.084,Y -551.105,Z 772.342,A 0.000,B 0.000,C 90.000,E1 277.473} C_DIS
LIN {X -0.102,Y -550.604,Z 772.335,A 0.000,B 0.000,C 90.000,E1 276.372} C_DIS
LIN {X 0.184,Y -549.918,Z 772.329,A 0.000,B 0.000,C 90.000,E1 275.220} C_DIS
LIN {X 0.047,Y -548.632,Z 772.318,A 0.000,B 0.000,C 90.000,E1 273.269} C_DIS
LIN {X -0.120,Y -547.496,Z 772.307,A 0.000,B 0.000,C 90.000,E1 271.318} C_DIS
LIN {X 0.153,Y -546.421,Z 772.298,A 0.000,B 0.000,C 90.000,E1 269.599} C_DIS
LIN {X -0.131,Y -545.261,Z 772.289,A 0.000,B 0.000,C 90.000,E1 267.936} C_DIS
LIN {X 0.074,Y -544.347,Z 772.281,A 0.000,B 0.000,C 90.000,E1 266.502} C_DIS
LIN {X -0.154,Y -543.133,Z 772.270,A 0.000,B 0.000,C 90.000,E1 264.546} C_DIS
LIN {X 0.027,Y -542.349,Z 772.263,A 0.000,B 0.000,C 90.000,E1 263.394} C_DIS
LIN {X 0.189,Y -541.387,Z 772.257,A 0.000,B 0.000,C 90.000,E1 262.243} C_DIS
LIN {X 0.001,Y -539.782,Z 772.246,A 0.000,B 0.000,C 90.000,E1 260.274} C_DIS
LIN {X 0.028,Y -537.818,Z 772.233,A 0.000,B 0.000,C 90.000,E1 257.993} C_DIS
LIN {X -0.182,Y -536.478,Z 772.225,A 0.000,B 0.000,C 90.000,E1 256.589} C_DIS
LIN {X 0.116,Y -535.661,Z 772.221,A 0.000,B 0.000,C 90.000,E1 255.700} C_DIS
LIN {X 0.174,Y -533.786,Z 772.211,A 0.000,B 0.000,C 90.000,E1 253.976} C_DIS
LIN {X 0.052,Y -531.208,Z 772.198,A 0.000,B 0.000,C 90.000,E1 251.692} C_DIS
LIN {X -0.227,Y -530.153,Z 772.194,A 0.000,B 0.000,C 90.000,E1 250.859} C_DIS
LIN {X 0.197,Y -527.716,Z 772.184,A 0.000,B 0.000,C 90.000,E1 249.082} C_DIS
LIN {X -0.093,Y -525.645,Z 772.176,A 0.000,B 0.000,C 90.000,E1 247.667} C_DIS
LIN {X -0.058,Y -522.999,Z 772.166,A 0.000,B 0.000,C 90.000,E1 245.921} C_DIS
LIN {X -0.016,Y -520.648,Z 772.158,A 0.000,B 0.000,C 90.000,E1 244.460} C_DIS
LIN {X -0.016,Y -518.253,Z 772.150,A 0.000,B 0.000,C 90.000,E1 242.999} C_DIS
LIN {X -0.194,Y -516.189,Z 772.143,A 0.000,B 0.000,C 90.000,E1 241.847} C_DIS
LIN {X -0.160,Y -513.932,Z 772.137,A 0.000,B 0.000,C 90.000,E1 240.667} C_DIS
LIN {X 0.086,Y -510.527,Z 772.127,A 0.000,B 0.000,C 90.000,E1 238.869} C_DIS
LIN {X -0.038,Y -508.785,Z 772.122,A 0.000,B 0.000,C 90.000,E1 237.995} C_DIS
LIN {X 0.139,Y -506.357,Z 772.116,A 0.000,B 0.000,C 90.000,E1 236.786} C_DIS
LIN {X 0.136,Y -503.760,Z 772.109,A 0.000,B 0.000,C 90.000,E1 235.595} C_DIS
LIN {X 0.099,Y -500.973,Z 772.102,A 0.000,B 0.000,C 90.000,E1 234.402} C_DIS
LIN {X -0.110,Y -497.237,Z 772.094,A 0.000,B 0.000,C 90.000,E1 232.924} C_DIS
LIN {X -0.229,Y -491.235,Z 772.081,A 0.000,B 0.000,C 90.000,E1 230.517} C_DIS
LIN {X -0.271,Y -485.561,Z 772.067,A 0.000,B 0.000,C 90.000,E1 228.081} C_DIS
LIN {X 0.173,Y -480.286,Z 772.053,A 0.000,B 0.000,C 90.000,E1 225.567} C_DIS
LIN {X 0.103,Y -476.924,Z 772.045,A 0.000,B 0.000,C 90.000,E1 224.028} C_DIS
LIN {X -0.011,Y -473.548,Z 772.036,A 0.000,B 0.000,C 90.000,E1 222.486} C_DIS
LIN {X -0.026,Y -468.767,Z 772.024,A 0.000,B 0.000,C 90.000,E1 220.297} C_DIS
LIN {X 0.170,Y -464.774,Z 772.013,A 0.000,B 0.000,C 90.000,E1 218.382} C_DIS
LIN {X -0.012,Y -460.766,Z 772.003,A 0.000,B 0.000,C 90.000,E1 216.503} C_DIS
LIN {X -0.028,Y -458.164,Z 771.996,A 0.000,B 0.000,C 90.000,E1 215.231} C_DIS
LIN {X 0.215,Y -453.605,Z 771.983,A 0.000,B 0.000,C 90.000,E1 212.959} C_DIS
LIN {X -0.084,Y -450.440,Z 771.974,A 0.000,B 0.000,C 90.000,E1 211.386} C_DIS
LIN {X 0.168,Y -446.766,Z 771.964,A 0.000,B 0.000,C 90.000,E1 209.411} C_DIS
LIN {X 0.175,Y -442.446,Z 771.951,A 0.000,B 0.000,C 90.000,E1 207.129} C_DIS
LIN {X 0.063,Y -438.129,Z 771.938,A 0.000,B 0.000,C 90.000,E1 204.847} C_DIS
LIN {X -0.172,Y -434.376,Z 771.927,A 0.000,B 0.000,C 90.000,E1 202.898} C_DIS
LIN {X 0.097,Y -431.873,Z 771.920,A 0.000,B 0.000,C 90.000,E1 201.535} C_DIS
LIN {X -0.022,Y -428.674,Z 771.911,A 0.000,B 0.000,C 90.000,E1 199.885} C_DIS
LIN {X 0.199,Y -425.493,Z 771.901,A 0.000,B 0.000,C 90.000,E1 198.181} C_DIS
LIN {X 0.031,Y -422.926,Z 771.894,A 0.000,B 0.000,C 90.000,E1 196.858} C_DIS
LIN {X 0.041,Y -418.937,Z 771.882,A 0.000,B 0.000,C 90.000,E1 194.828} C_DIS
LIN {X -0.206,Y -414.482,Z 771.869,A 0.000,B 0.000,C 90.000,E1 192.479} C_DIS
LIN {X -0.173,Y -410.226,Z 771.856,A 0.000,B 0.000,C 90.000,E1 190.074} C_DIS
LIN {X -0.090,Y -406.672,Z 771.844,A 0.000,B 0.000,C 90.000,E1 187.992} C_DIS
LIN {X -0.134,Y -402.631,Z 771.831,A 0.000,B 0.000,C 90.000,E1 185.568} C_DIS
LIN {X 0.003,Y -398.307,Z 771.815,A 0.000,B 0.000,C 90.000,E1 182.751} C_DIS
LIN {X -0.122,Y -394.227,Z 771.798,A 0.000,B 0.000,C 90.000,E1 179.599} C_DIS
LIN {X 0.016,Y -390.718,Z 771.780,A 0.000,B 0.000,C 90.000,E1 176.388} C_DIS
LIN {X -0.053,Y -388.796,Z 771.768,A 0.000,B 0.000,C 90.000,E1 174.261} C_DIS
LIN {X 0.048,Y -386.172,Z 771.750,A 0.000,B 0.000,C 90.000,E1 171.027} C_DIS
LIN {X 0.075,Y -384.658,Z 771.738,A 0.000,B 0.000,C 90.000,E1 168.870} C_DIS
LIN {X 0.144,Y -383.533,Z 771.728,A 0.000,B 0.000,C 90.000,E1 167.061} C_DIS
LIN {X -0.105,Y -382.516,Z 771.716,A 0.000,B 0.000,C 90.000,E1 164.936} C_DIS
LIN {X -0.162,Y -381.502,Z 771.702,A 0.000,B 0.000,C 90.000,E1 162.417} C_DIS
LIN {X 0.010,Y -380.601,Z 771.684,A 0.000,B 0.000,C 90.000,E1 159.135} C_DIS
LIN {X -0.076,Y -380.318,Z 771.670,A 0.000,B 0.000,C 90.000,E1 156.613} C_DIS
LIN {X -0.081,Y -380.774,Z 771.654,A 0.000,B 0.000,C 90.000,E1 153.717} C_DIS
LIN {X 0.135,Y -381.533,Z 771.642,A 0.000,B 0.000,C 90.000,E1 151.513} C_DIS
LIN {X -0.114,Y -382.698,Z 771.632,A 0.000,B 0.000,C 90.000,E1 149.744} C_DIS
LIN {X 0.033,Y -385.404,Z 771.618,A 0.000,B 0.000,C 90.000,E1 147.199} C_DIS
LIN {X 0.149,Y -387.902,Z 771.608,A 0.000,B 0.000,C 90.000,E1 145.388} C_DIS
LIN {X 0.103,Y -389.997,Z 771.602,A 0.000,B 0.000,C 90.000,E1 144.322} C_DIS
LIN {X 0.009,Y -391.574,Z 771.598,A 0.000,B 0.000,C 90.000,E1 143.623} C_DIS
LIN {X -0.074,Y -393.404,Z 771.594,A 0.000,B 0.000,C 90.000,E1 142.924} C_DIS
LIN {X 0.094,Y -395.711,Z 771.590,A 0.000,B 0.000,C 90.000,E1 142.190} C_DIS
LIN {X 0.040,Y -398.726,Z 771.586,A 0.000,B 0.000,C 90.000,E1 141.492} C_DIS
LIN {X -0.103,Y -401.867,Z 771.583,A 0.000,B 0.000,C 90.000,E1 140.928} C_DIS
LIN {X 0.162,Y -404.756,Z 771.580,A 0.000,B 0.000,C 90.000,E1 140.436} C_DIS
LIN {X 0.163,Y -409.346,Z 771.577,A 0.000,B 0.000,C 90.000,E1 139.828} C_DIS
LIN {X -0.177,Y -414.966,Z 771.573,A 0.000,B 0.000,C 90.000,E1 139.218} C_DIS
LIN {X 0.094,Y -422.103,Z 771.569,A 0.000,B 0.000,C 90.000,E1 138.405} C_DIS
LIN {X 0.053,Y -437.952,Z 771.560,A 0.000,B 0.000,C 90.000,E1 136.743} C_DIS
LIN {X 0.237,Y -444.978,Z 771.556,A 0.000,B 0.000,C 90.000,E1 135.972} C_DIS
LIN {X -0.051,Y -454.628,Z 771.550,A 0.000,B 0.000,C 90.000,E1 134.960} C_DIS
LIN {X -0.084,Y -460.051,Z 771.546,A 0.000,B 0.000,C 90.000,E1 134.352} C_DIS
LIN {X 0.120,Y -465.301,Z 771.543,A 0.000,B 0.000,C 90.000,E1 133.704} C_DIS
LIN {X 0.047,Y -474.327,Z 771.537,A 0.000,B 0.000,C 90.000,E1 132.609} C_DIS
LIN {X 0.188,Y -480.356,Z 771.533,A 0.000,B 0.000,C 90.000,E1 131.838} C_DIS
LIN {X 0.111,Y -485.079,Z 771.529,A 0.000,B 0.000,C 90.000,E1 131.229} C_DIS
LIN {X 0.068,Y -489.568,Z 771.526,A 0.000,B 0.000,C 90.000,E1 130.620} C_DIS
LIN {X -0.023,Y -492.830,Z 771.523,A 0.000,B 0.000,C 90.000,E1 130.172} C_DIS
LIN {X -0.070,Y -498.931,Z 771.518,A 0.000,B 0.000,C 90.000,E1 129.277} C_DIS
LIN {X -0.103,Y -504.619,Z 771.513,A 0.000,B 0.000,C 90.000,E1 128.382} C_DIS
LIN {X -0.321,Y -508.258,Z 771.510,A 0.000,B 0.000,C 90.000,E1 127.810} C_DIS
LIN {X 0.008,Y -512.500,Z 771.506,A 0.000,B 0.000,C 90.000,E1 127.030} C_DIS
LIN {X -0.102,Y -518.212,Z 771.500,A 0.000,B 0.000,C 90.000,E1 126.011} C_DIS
LIN {X -0.144,Y -522.733,Z 771.495,A 0.000,B 0.000,C 90.000,E1 125.152} C_DIS
LIN {X 0.196,Y -525.628,Z 771.492,A 0.000,B 0.000,C 90.000,E1 124.532} C_DIS
LIN {X -0.001,Y -529.470,Z 771.487,A 0.000,B 0.000,C 90.000,E1 123.706} C_DIS
LIN {X 0.224,Y -533.788,Z 771.482,A 0.000,B 0.000,C 90.000,E1 122.673} C_DIS
LIN {X 0.215,Y -537.915,Z 771.476,A 0.000,B 0.000,C 90.000,E1 121.671} C_DIS
LIN {X 0.123,Y -542.142,Z 771.470,A 0.000,B 0.000,C 90.000,E1 120.541} C_DIS
LIN {X -0.125,Y -545.093,Z 771.465,A 0.000,B 0.000,C 90.000,E1 119.716} C_DIS
LIN {X 0.091,Y -548.811,Z 771.459,A 0.000,B 0.000,C 90.000,E1 118.565} C_DIS
LIN {X -0.113,Y -552.301,Z 771.453,A 0.000,B 0.000,C 90.000,E1 117.462} C_DIS
LIN {X -0.049,Y -554.571,Z 771.448,A 0.000,B 0.000,C 90.000,E1 116.616} C_DIS
LIN {X 0.006,Y -555.832,Z 771.445,A 0.000,B 0.000,C 90.000,E1 116.052} C_DIS
LIN {X -0.113,Y -558.087,Z 771.439,A 0.000,B 0.000,C 90.000,E1 114.951} C_DIS
LIN {X 0.062,Y -559.729,Z 771.432,A 0.000,B 0.000,C 90.000,E1 113.823} C_DIS
LIN {X -0.054,Y -562.263,Z 771.422,A 0.000,B 0.000,C 90.000,E1 111.897} C_DIS
LIN {X 0.288,Y -563.794,Z 771.414,A 0.000,B 0.000,C 90.000,E1 110.482} C_DIS
LIN {X -0.071,Y -565.249,Z 771.406,A 0.000,B 0.000,C 90.000,E1 109.141} C_DIS
LIN {X 0.277,Y -566.696,Z 771.397,A 0.000,B 0.000,C 90.000,E1 107.457} C_DIS
LIN {X 0.120,Y -568.354,Z 771.387,A 0.000,B 0.000,C 90.000,E1 105.552} C_DIS
LIN {X -0.180,Y -569.719,Z 771.377,A 0.000,B 0.000,C 90.000,E1 103.939} C_DIS
LIN {X 0.010,Y -571.466,Z 771.367,A 0.000,B 0.000,C 90.000,E1 102.007} C_DIS
LIN {X -0.221,Y -573.487,Z 771.355,A 0.000,B 0.000,C 90.000,E1 99.849} C_DIS
LIN {X 0.120,Y -574.610,Z 771.347,A 0.000,B 0.000,C 90.000,E1 98.454} C_DIS
LIN {X -0.172,Y -575.726,Z 771.340,A 0.000,B 0.000,C 90.000,E1 97.125} C_DIS
LIN {X 0.124,Y -576.656,Z 771.332,A 0.000,B 0.000,C 90.000,E1 95.739} C_DIS
LIN {X 0.228,Y -577.356,Z 771.326,A 0.000,B 0.000,C 90.000,E1 94.645} C_DIS
LIN {X 0.063,Y -578.414,Z 771.317,A 0.000,B 0.000,C 90.000,E1 93.037} C_DIS
LIN {X -0.113,Y -579.249,Z 771.308,A 0.000,B 0.000,C 90.000,E1 91.432} C_DIS
LIN {X -0.280,Y -580.025,Z 771.299,A 0.000,B 0.000,C 90.000,E1 89.828} C_DIS
LIN {X -0.189,Y -580.462,Z 771.293,A 0.000,B 0.000,C 90.000,E1 88.740} C_DIS
LIN {X 0.258,Y -580.996,Z 771.284,A 0.000,B 0.000,C 90.000,E1 87.078} C_DIS
LIN {X 0.002,Y -581.383,Z 771.276,A 0.000,B 0.000,C 90.000,E1 85.755} C_DIS
LIN {X -0.079,Y -581.688,Z 771.268,A 0.000,B 0.000,C 90.000,E1 84.147} C_DIS
LIN {X -0.032,Y -581.881,Z 771.258,A 0.000,B 0.000,C 90.000,E1 82.527} C_DIS
LIN {X -0.202,Y -581.956,Z 771.251,A 0.000,B 0.000,C 90.000,E1 81.197} C_DIS
LIN {X 0.289,Y -582.064,Z 771.244,A 0.000,B 0.000,C 90.000,E1 79.803} C_DIS
LIN {X 0.202,Y -582.023,Z 771.236,A 0.000,B 0.000,C 90.000,E1 78.465} C_DIS
LIN {X 0.120,Y -581.676,Z 771.226,A 0.000,B 0.000,C 90.000,E1 76.589} C_DIS
LIN {X 0.271,Y -581.262,Z 771.218,A 0.000,B 0.000,C 90.000,E1 75.227} C_DIS
LIN {X -0.143,Y -580.781,Z 771.211,A 0.000,B 0.000,C 90.000,E1 73.921} C_DIS
LIN {X -0.192,Y -580.170,Z 771.202,A 0.000,B 0.000,C 90.000,E1 72.308} C_DIS
LIN {X -0.083,Y -579.372,Z 771.193,A 0.000,B 0.000,C 90.000,E1 70.678} C_DIS
LIN {X 0.201,Y -578.432,Z 771.184,A 0.000,B 0.000,C 90.000,E1 69.028} C_DIS
LIN {X -0.089,Y -577.666,Z 771.178,A 0.000,B 0.000,C 90.000,E1 67.975} C_DIS
LIN {X -0.160,Y -576.368,Z 771.169,A 0.000,B 0.000,C 90.000,E1 66.357} C_DIS
LIN {X 0.281,Y -575.365,Z 771.163,A 0.000,B 0.000,C 90.000,E1 65.229} C_DIS
LIN {X 0.027,Y -573.919,Z 771.155,A 0.000,B 0.000,C 90.000,E1 63.896} C_DIS
LIN {X -0.096,Y -572.546,Z 771.149,A 0.000,B 0.000,C 90.000,E1 62.820} C_DIS
LIN {X 0.018,Y -570.944,Z 771.143,A 0.000,B 0.000,C 90.000,E1 61.719} C_DIS
LIN {X -0.111,Y -569.082,Z 771.137,A 0.000,B 0.000,C 90.000,E1 60.639} C_DIS
LIN {X -0.045,Y -567.018,Z 771.131,A 0.000,B 0.000,C 90.000,E1 59.537} C_DIS
LIN {X -0.213,Y -564.590,Z 771.125,A 0.000,B 0.000,C 90.000,E1 58.456} C_DIS
LIN {X 0.267,Y -562.505,Z 771.120,A 0.000,B 0.000,C 90.000,E1 57.582} C_DIS
LIN {X -0.058,Y -560.251,Z 771.115,A 0.000,B 0.000,C 90.000,E1 56.786} C_DIS
LIN {X -0.102,Y -557.801,Z 771.111,A 0.000,B 0.000,C 90.000,E1 55.960} C_DIS
LIN {X 0.064,Y -556.086,Z 771.108,A 0.000,B 0.000,C 90.000,E1 55.388} C_DIS
LIN {X -0.025,Y -553.245,Z 771.103,A 0.000,B 0.000,C 90.000,E1 54.562} C_DIS
LIN {X 0.113,Y -551.164,Z 771.100,A 0.000,B 0.000,C 90.000,E1 53.989} C_DIS
LIN {X 0.290,Y -547.684,Z 771.095,A 0.000,B 0.000,C 90.000,E1 53.130} C_DIS
LIN {X -0.192,Y -544.528,Z 771.091,A 0.000,B 0.000,C 90.000,E1 52.477} C_DIS
LIN {X 0.064,Y -541.066,Z 771.088,A 0.000,B 0.000,C 90.000,E1 51.743} C_DIS
LIN {X 0.109,Y -538.153,Z 771.084,A 0.000,B 0.000,C 90.000,E1 51.170} C_DIS
LIN {X 0.128,Y -534.931,Z 771.081,A 0.000,B 0.000,C 90.000,E1 50.598} C_DIS
LIN {X -0.039,Y -530.428,Z 771.077,A 0.000,B 0.000,C 90.000,E1 49.908} C_DIS
LIN {X 0.262,Y -526.383,Z 771.074,A 0.000,B 0.000,C 90.000,E1 49.299} C_DIS
LIN {X -0.132,Y -521.825,Z 771.071,A 0.000,B 0.000,C 90.000,E1 48.771} C_DIS
LIN {X 0.200,Y -516.915,Z 771.068,A 0.000,B 0.000,C 90.000,E1 48.162} C_DIS
LIN {X -0.013,Y -512.934,Z 771.065,A 0.000,B 0.000,C 90.000,E1 47.757} C_DIS
LIN {X -0.249,Y -507.180,Z 771.062,A 0.000,B 0.000,C 90.000,E1 47.229} C_DIS
LIN {X -0.160,Y -502.848,Z 771.060,A 0.000,B 0.000,C 90.000,E1 46.824} C_DIS
LIN {X -0.281,Y -495.196,Z 771.057,A 0.000,B 0.000,C 90.000,E1 46.215} C_DIS
LIN {X 0.139,Y -487.469,Z 771.053,A 0.000,B 0.000,C 90.000,E1 45.567} C_DIS
LIN {X 0.123,Y -479.397,Z 771.050,A 0.000,B 0.000,C 90.000,E1 45.000} C_DIS
LIN {X -0.221,Y -471.533,Z 771.047,A 0.000,B 0.000,C 90.000,E1 44.514} C_DIS
LIN {X -0.166,Y -461.843,Z 771.044,A 0.000,B 0.000,C 90.000,E1 43.866} C_DIS
LIN {X 0.105,Y -442.419,Z 771.036,A 0.000,B 0.000,C 90.000,E1 42.528} C_DIS
LIN {X 0.158,Y -423.232,Z 771.029,A 0.000,B 0.000,C 90.000,E1 41.148} C_DIS
LIN {X -0.101,Y -414.073,Z 771.025,A 0.000,B 0.000,C 90.000,E1 40.458} C_DIS
LIN {X -0.159,Y -408.256,Z 771.022,A 0.000,B 0.000,C 90.000,E1 39.930} C_DIS
LIN {X 0.123,Y -408.224,Z 771.022,A 0.000,B 0.000,C 90.000,E1 39.886} C_DIS
LIN {X -0.253,Y -405.740,Z 771.014,A 0.000,B 0.000,C 90.000,E1 38.463} C_DIS
LIN {X -0.029,Y -398.664,Z 770.994,A 0.000,B 0.000,C 90.000,E1 34.945} C_DIS
LIN {X -0.040,Y -398.437,Z 770.993,A 0.000,B 0.000,C 90.000,E1 34.771} C_DIS
LIN {X 0.092,Y -399.151,Z 770.975,A 0.000,B 0.000,C 90.000,E1 31.416} C_DIS
LIN {X -0.058,Y -400.505,Z 770.957,A 0.000,B 0.000,C 90.000,E1 28.281} C_DIS
LIN {X 0.077,Y -402.162,Z 770.942,A 0.000,B 0.000,C 90.000,E1 25.463} C_DIS
LIN {X 0.012,Y -404.404,Z 770.924,A 0.000,B 0.000,C 90.000,E1 22.333} C_DIS
LIN {X 0.076,Y -407.759,Z 770.905,A 0.000,B 0.000,C 90.000,E1 18.852} C_DIS
LIN {X 0.022,Y -412.754,Z 770.884,A 0.000,B 0.000,C 90.000,E1 15.064} C_DIS
LIN {X 0.162,Y -416.420,Z 770.870,A 0.000,B 0.000,C 90.000,E1 12.647} C_DIS
LIN {X 0.106,Y -419.223,Z 770.861,A 0.000,B 0.000,C 90.000,E1 10.950} C_DIS
LIN {X 0.104,Y -422.645,Z 770.850,A 0.000,B 0.000,C 90.000,E1 8.916} C_DIS
LIN {X 0.031,Y -425.550,Z 770.840,A 0.000,B 0.000,C 90.000,E1 7.239} C_DIS
LIN {X 0.218,Y -430.198,Z 770.825,A 0.000,B 0.000,C 90.000,E1 4.531} C_DIS
LIN {X 0.031,Y -435.153,Z 770.811,A 0.000,B 0.000,C 90.000,E1 1.892} C_DIS
LIN {X -0.162,Y -439.959,Z 770.797,A 0.000,B 0.000,C 90.000,E1 359.484} C_DIS
LIN {X -0.037,Y -445.426,Z 770.782,A 0.000,B 0.000,C 90.000,E1 356.846} C_DIS
LIN {X 0.106,Y -450.678,Z 770.770,A 0.000,B 0.000,C 90.000,E1 354.552} C_DIS
LIN {X 0.148,Y -454.465,Z 770.761,A 0.000,B 0.000,C 90.000,E1 352.932} C_DIS
LIN {X 0.052,Y -457.409,Z 770.754,A 0.000,B 0.000,C 90.000,E1 351.659} C_DIS
LIN {X -0.004,Y -460.313,Z 770.747,A 0.000,B 0.000,C 90.000,E1 350.387} C_DIS
LIN {X 0.057,Y -463.044,Z 770.740,A 0.000,B 0.000,C 90.000,E1 349.106} C_DIS
LIN {X -0.065,Y -468.530,Z 770.726,A 0.000,B 0.000,C 90.000,E1 346.589} C_DIS
LIN {X 0.127,Y -470.341,Z 770.722,A 0.000,B 0.000,C 90.000,E1 345.936} C_DIS
LIN {X 0.161,Y -472.145,Z 770.719,A 0.000,B 0.000,C 90.000,E1 345.463} C_DIS
LIN {X 0.060,Y -474.028,Z 770.717,A 0.000,B 0.000,C 90.000,E1 345.102} C_DIS
LIN {X 0.094,Y -477.055,Z 770.715,A 0.000,B 0.000,C 90.000,E1 344.629} C_DIS
LIN {X -0.110,Y -480.056,Z 770.713,A 0.000,B 0.000,C 90.000,E1 344.283} C_DIS
LIN {X 0.266,Y -487.049,Z 770.709,A 0.000,B 0.000,C 90.000,E1 343.559} C_DIS
LIN {X 0.161,Y -494.981,Z 770.706,A 0.000,B 0.000,C 90.000,E1 342.960} C_DIS
LIN {X 0.231,Y -516.917,Z 770.697,A 0.000,B 0.000,C 90.000,E1 341.456} C_DIS
LIN {X -0.048,Y -537.364,Z 770.690,A 0.000,B 0.000,C 90.000,E1 340.188} C_DIS
LIN {X 0.269,Y -543.549,Z 770.688,A 0.000,B 0.000,C 90.000,E1 339.752} C_DIS
LIN {X 0.186,Y -547.988,Z 770.686,A 0.000,B 0.000,C 90.000,E1 339.444} C_DIS
LIN {X -0.156,Y -553.663,Z 770.683,A 0.000,B 0.000,C 90.000,E1 339.028} C_DIS
LIN {X -0.027,Y -560.324,Z 770.680,A 0.000,B 0.000,C 90.000,E1 338.411} C_DIS
LIN {X -0.252,Y -565.449,Z 770.677,A 0.000,B 0.000,C 90.000,E1 337.922} C_DIS
LIN {X 0.142,Y -570.333,Z 770.674,A 0.000,B 0.000,C 90.000,E1 337.358} C_DIS
LIN {X -0.097,Y -573.973,Z 770.672,A 0.000,B 0.000,C 90.000,E1 336.975} C_DIS
LIN {X -0.346,Y -581.769,Z 770.667,A 0.000,B 0.000,C 90.000,E1 336.049} C_DIS
LIN {X -0.272,Y -588.860,Z 770.662,A 0.000,B 0.000,C 90.000,E1 335.101} C_DIS
LIN {X -0.108,Y -595.515,Z 770.656,A 0.000,B 0.000,C 90.000,E1 334.152} C_DIS
LIN {X 0.174,Y -601.153,Z 770.652,A 0.000,B 0.000,C 90.000,E1 333.332} C_DIS
LIN {X 0.002,Y -605.512,Z 770.648,A 0.000,B 0.000,C 90.000,E1 332.692} C_DIS
LIN {X 0.086,Y -612.178,Z 770.643,A 0.000,B 0.000,C 90.000,E1 331.641} C_DIS
LIN {X 0.281,Y -617.732,Z 770.638,A 0.000,B 0.000,C 90.000,E1 330.717} C_DIS
LIN {X 0.005,Y -625.375,Z 770.630,A 0.000,B 0.000,C 90.000,E1 329.459} C_DIS
LIN {X -0.173,Y -630.939,Z 770.625,A 0.000,B 0.000,C 90.000,E1 328.456} C_DIS
LIN {X -0.282,Y -636.282,Z 770.619,A 0.000,B 0.000,C 90.000,E1 327.454} C_DIS
LIN {X -0.001,Y -640.547,Z 770.614,A 0.000,B 0.000,C 90.000,E1 326.548} C_DIS
LIN {X -0.124,Y -646.311,Z 770.607,A 0.000,B 0.000,C 90.000,E1 325.308} C_DIS
LIN {X 0.306,Y -650.525,Z 770.602,A 0.000,B 0.000,C 90.000,E1 324.276} C_DIS
LIN {X 0.197,Y -653.549,Z 770.598,A 0.000,B 0.000,C 90.000,E1 323.543} C_DIS
LIN {X 0.190,Y -657.342,Z 770.592,A 0.000,B 0.000,C 90.000,E1 322.557} C_DIS
LIN {X -0.298,Y -660.886,Z 770.587,A 0.000,B 0.000,C 90.000,E1 321.618} C_DIS
LIN {X 0.163,Y -665.043,Z 770.580,A 0.000,B 0.000,C 90.000,E1 320.356} C_DIS
LIN {X 0.199,Y -667.380,Z 770.576,A 0.000,B 0.000,C 90.000,E1 319.622} C_DIS
LIN {X -0.250,Y -670.460,Z 770.570,A 0.000,B 0.000,C 90.000,E1 318.690} C_DIS
LIN {X -0.142,Y -673.887,Z 770.564,A 0.000,B 0.000,C 90.000,E1 317.472} C_DIS
LIN {X -0.013,Y -676.862,Z 770.557,A 0.000,B 0.000,C 90.000,E1 316.257} C_DIS
LIN {X -0.341,Y -679.075,Z 770.552,A 0.000,B 0.000,C 90.000,E1 315.324} C_DIS
LIN {X -0.125,Y -681.538,Z 770.545,A 0.000,B 0.000,C 90.000,E1 314.109} C_DIS
LIN {X -0.343,Y -683.778,Z 770.538,A 0.000,B 0.000,C 90.000,E1 312.933} C_DIS
LIN {X 0.384,Y -685.466,Z 770.533,A 0.000,B 0.000,C 90.000,E1 311.919} C_DIS
LIN {X 0.161,Y -686.987,Z 770.528,A 0.000,B 0.000,C 90.000,E1 310.987} C_DIS
LIN {X -0.112,Y -687.989,Z 770.524,A 0.000,B 0.000,C 90.000,E1 310.297} C_DIS
LIN {X -0.168,Y -689.427,Z 770.517,A 0.000,B 0.000,C 90.000,E1 309.116} C_DIS
LIN {X -0.023,Y -691.039,Z 770.509,A 0.000,B 0.000,C 90.000,E1 307.684} C_DIS
LIN {X -0.035,Y -692.146,Z 770.503,A 0.000,B 0.000,C 90.000,E1 306.503} C_DIS
LIN {X 0.110,Y -693.192,Z 770.496,A 0.000,B 0.000,C 90.000,E1 305.311} C_DIS
LIN {X 0.272,Y -694.098,Z 770.490,A 0.000,B 0.000,C 90.000,E1 304.119} C_DIS
LIN {X -0.052,Y -695.353,Z 770.481,A 0.000,B 0.000,C 90.000,E1 302.498} C_DIS
LIN {X 0.007,Y -696.459,Z 770.473,A 0.000,B 0.000,C 90.000,E1 301.082} C_DIS
LIN {X -0.180,Y -697.222,Z 770.466,A 0.000,B 0.000,C 90.000,E1 299.922} C_DIS
LIN {X 0.059,Y -697.973,Z 770.456,A 0.000,B 0.000,C 90.000,E1 298.025} C_DIS
LIN {X -0.053,Y -698.908,Z 770.444,A 0.000,B 0.000,C 90.000,E1 295.924} C_DIS
LIN {X -0.277,Y -699.594,Z 770.438,A 0.000,B 0.000,C 90.000,E1 294.771} C_DIS
LIN {X 0.258,Y -699.346,Z 770.435,A 0.000,B 0.000,C 90.000,E1 294.259} C_DIS
LIN {X 0.239,Y -699.120,Z 770.434,A 0.000,B 0.000,C 90.000,E1 294.027} C_DIS
LIN {X 0.128,Y -697.659,Z 770.431,A 0.000,B 0.000,C 90.000,E1 293.567} C_DIS
LIN {X 0.111,Y -696.684,Z 770.430,A 0.000,B 0.000,C 90.000,E1 293.334} C_DIS
LIN {X 0.240,Y -695.789,Z 770.429,A 0.000,B 0.000,C 90.000,E1 293.206} C_DIS
LIN {X -0.127,Y -693.300,Z 770.428,A 0.000,B 0.000,C 90.000,E1 293.003} C_DIS
LIN {X -0.012,Y -690.634,Z 770.427,A 0.000,B 0.000,C 90.000,E1 292.770} C_DIS
LIN {X 0.229,Y -689.111,Z 770.426,A 0.000,B 0.000,C 90.000,E1 292.642} C_DIS
LIN {X -0.328,Y -686.880,Z 770.425,A 0.000,B 0.000,C 90.000,E1 292.589} C_DIS
LIN {X 0.013,Y -684.232,Z 770.425,A 0.000,B 0.000,C 90.000,E1 292.461} C_DIS
LIN {X 0.031,Y -679.920,Z 770.424,A 0.000,B 0.000,C 90.000,E1 292.333} C_DIS
LIN {X -0.045,Y -674.796,Z 770.423,A 0.000,B 0.000,C 90.000,E1 292.206} C_DIS
LIN {X -0.147,Y -666.206,Z 770.423,A 0.000,B 0.000,C 90.000,E1 292.078} C_DIS
LIN {X -0.054,Y -656.948,Z 770.422,A 0.000,B 0.000,C 90.000,E1 291.950} C_DIS
LIN {X 0.099,Y -643.603,Z 770.421,A 0.000,B 0.000,C 90.000,E1 291.716} C_DIS
LIN {X 0.218,Y -627.125,Z 770.419,A 0.000,B 0.000,C 90.000,E1 291.354} C_DIS
LIN {X -0.180,Y -609.707,Z 770.416,A 0.000,B 0.000,C 90.000,E1 290.972} C_DIS
LIN {X 0.124,Y -592.409,Z 770.414,A 0.000,B 0.000,C 90.000,E1 290.482} C_DIS
LIN {X 0.225,Y -568.242,Z 770.410,A 0.000,B 0.000,C 90.000,E1 289.758} C_DIS
LIN {X -0.092,Y -565.103,Z 770.409,A 0.000,B 0.000,C 90.000,E1 289.685} C_DIS
LIN {X 0.218,Y -559.107,Z 770.408,A 0.000,B 0.000,C 90.000,E1 289.396} C_DIS
LIN {X -0.254,Y -556.699,Z 770.407,A 0.000,B 0.000,C 90.000,E1 289.214} C_DIS
LIN {X 0.281,Y -555.781,Z 770.405,A 0.000,B 0.000,C 90.000,E1 288.906} C_DIS
LIN {X 0.252,Y -555.132,Z 770.402,A 0.000,B 0.000,C 90.000,E1 288.362} C_DIS
LIN {X 0.096,Y -554.495,Z 770.394,A 0.000,B 0.000,C 90.000,E1 286.985} C_DIS
LIN {X 0.136,Y -553.320,Z 770.379,A 0.000,B 0.000,C 90.000,E1 284.189} C_DIS
LIN {X -0.203,Y -552.800,Z 770.371,A 0.000,B 0.000,C 90.000,E1 282.827} C_DIS
LIN {X -0.138,Y -552.353,Z 770.363,A 0.000,B 0.000,C 90.000,E1 281.422} C_DIS
LIN {X 0.030,Y -551.745,Z 770.354,A 0.000,B 0.000,C 90.000,E1 279.726} C_DIS
LIN {X 0.109,Y -551.181,Z 770.343,A 0.000,B 0.000,C 90.000,E1 277.757} C_DIS
LIN {X -0.145,Y -550.716,Z 770.337,A 0.000,B 0.000,C 90.000,E1 276.663} C_DIS
LIN {X 0.147,Y -550.107,Z 770.331,A 0.000,B 0.000,C 90.000,E1 275.511} C_DIS
LIN {X 0.059,Y -548.768,Z 770.320,A 0.000,B 0.000,C 90.000,E1 273.555} C_DIS
LIN {X -0.108,Y -547.633,Z 770.309,A 0.000,B 0.000,C 90.000,E1 271.604} C_DIS
LIN {X 0.077,Y -546.975,Z 770.303,A 0.000,B 0.000,C 90.000,E1 270.458} C_DIS
LIN {X -0.248,Y -546.061,Z 770.295,A 0.000,B 0.000,C 90.000,E1 269.083} C_DIS
LIN {X 0.037,Y -544.707,Z 770.284,A 0.000,B 0.000,C 90.000,E1 267.078} C_DIS
LIN {X 0.258,Y -543.827,Z 770.276,A 0.000,B 0.000,C 90.000,E1 265.641} C_DIS
LIN {X -0.076,Y -542.954,Z 770.268,A 0.000,B 0.000,C 90.000,E1 264.261} C_DIS
LIN {X 0.170,Y -541.905,Z 770.260,A 0.000,B 0.000,C 90.000,E1 262.818} C_DIS
LIN {X 0.078,Y -540.015,Z 770.248,A 0.000,B 0.000,C 90.000,E1 260.557} C_DIS
LIN {X -0.257,Y -538.997,Z 770.241,A 0.000,B 0.000,C 90.000,E1 259.454} C_DIS
LIN {X 0.152,Y -537.591,Z 770.232,A 0.000,B 0.000,C 90.000,E1 257.701} C_DIS
LIN {X 0.120,Y -536.019,Z 770.222,A 0.000,B 0.000,C 90.000,E1 255.992} C_DIS
LIN {X 0.235,Y -533.824,Z 770.211,A 0.000,B 0.000,C 90.000,E1 253.976} C_DIS
LIN {X 0.112,Y -531.244,Z 770.198,A 0.000,B 0.000,C 90.000,E1 251.692} C_DIS
LIN {X -0.167,Y -530.191,Z 770.194,A 0.000,B 0.000,C 90.000,E1 250.859} C_DIS
LIN {X 0.259,Y -527.752,Z 770.184,A 0.000,B 0.000,C 90.000,E1 249.082} C_DIS
LIN {X -0.031,Y -525.692,Z 770.176,A 0.000,B 0.000,C 90.000,E1 247.667} C_DIS
LIN {X -0.156,Y -523.498,Z 770.168,A 0.000,B 0.000,C 90.000,E1 246.230} C_DIS
LIN {X -0.002,Y -521.655,Z 770.161,A 0.000,B 0.000,C 90.000,E1 245.049} C_DIS
LIN {X 0.008,Y -519.278,Z 770.153,A 0.000,B 0.000,C 90.000,E1 243.589} C_DIS
LIN {X -0.282,Y -517.788,Z 770.148,A 0.000,B 0.000,C 90.000,E1 242.743} C_DIS
LIN {X -0.129,Y -516.232,Z 770.144,A 0.000,B 0.000,C 90.000,E1 241.847} C_DIS
LIN {X -0.095,Y -513.960,Z 770.137,A 0.000,B 0.000,C 90.000,E1 240.667} C_DIS
LIN {X 0.151,Y -510.548,Z 770.127,A 0.000,B 0.000,C 90.000,E1 238.869} C_DIS
LIN {X 0.027,Y -508.811,Z 770.122,A 0.000,B 0.000,C 90.000,E1 237.995} C_DIS
LIN {X -0.218,Y -506.420,Z 770.116,A 0.000,B 0.000,C 90.000,E1 236.834} C_DIS
LIN {X 0.201,Y -503.816,Z 770.109,A 0.000,B 0.000,C 90.000,E1 235.595} C_DIS
LIN {X 0.048,Y -500.307,Z 770.101,A 0.000,B 0.000,C 90.000,E1 234.116} C_DIS
LIN {X -0.043,Y -497.302,Z 770.094,A 0.000,B 0.000,C 90.000,E1 232.924} C_DIS
LIN {X -0.161,Y -491.281,Z 770.081,A 0.000,B 0.000,C 90.000,E1 230.517} C_DIS
LIN {X -0.027,Y -486.289,Z 770.069,A 0.000,B 0.000,C 90.000,E1 228.366} C_DIS
LIN {X 0.042,Y -482.890,Z 770.060,A 0.000,B 0.000,C 90.000,E1 226.824} C_DIS
LIN {X 0.031,Y -479.645,Z 770.052,A 0.000,B 0.000,C 90.000,E1 225.283} C_DIS
LIN {X 0.285,Y -476.263,Z 770.043,A 0.000,B 0.000,C 90.000,E1 223.704} C_DIS
LIN {X 0.059,Y -473.581,Z 770.036,A 0.000,B 0.000,C 90.000,E1 222.486} C_DIS
LIN {X 0.115,Y -470.831,Z 770.029,A 0.000,B 0.000,C 90.000,E1 221.229} C_DIS
LIN {X 0.239,Y -467.474,Z 770.020,A 0.000,B 0.000,C 90.000,E1 219.644} C_DIS
LIN {X 0.241,Y -464.837,Z 770.013,A 0.000,B 0.000,C 90.000,E1 218.382} C_DIS
LIN {X -0.193,Y -460.172,Z 770.001,A 0.000,B 0.000,C 90.000,E1 216.217} C_DIS
LIN {X -0.001,Y -456.236,Z 769.990,A 0.000,B 0.000,C 90.000,E1 214.278} C_DIS
LIN {X 0.100,Y -452.384,Z 769.980,A 0.000,B 0.000,C 90.000,E1 212.339} C_DIS
LIN {X 0.168,Y -447.455,Z 769.965,A 0.000,B 0.000,C 90.000,E1 209.745} C_DIS
LIN {X -0.194,Y -443.145,Z 769.953,A 0.000,B 0.000,C 90.000,E1 207.513} C_DIS
LIN {X -0.099,Y -438.830,Z 769.940,A 0.000,B 0.000,C 90.000,E1 205.207} C_DIS
LIN {X 0.075,Y -435.067,Z 769.929,A 0.000,B 0.000,C 90.000,E1 203.206} C_DIS
LIN {X -0.049,Y -432.610,Z 769.922,A 0.000,B 0.000,C 90.000,E1 201.897} C_DIS
LIN {X 0.059,Y -428.752,Z 769.911,A 0.000,B 0.000,C 90.000,E1 199.885} C_DIS
LIN {X -0.125,Y -425.560,Z 769.901,A 0.000,B 0.000,C 90.000,E1 198.236} C_DIS
LIN {X 0.112,Y -423.010,Z 769.894,A 0.000,B 0.000,C 90.000,E1 196.858} C_DIS
LIN {X -0.101,Y -420.361,Z 769.886,A 0.000,B 0.000,C 90.000,E1 195.536} C_DIS
LIN {X -0.123,Y -414.580,Z 769.869,A 0.000,B 0.000,C 90.000,E1 192.479} C_DIS
LIN {X -0.087,Y -410.324,Z 769.856,A 0.000,B 0.000,C 90.000,E1 190.074} C_DIS
LIN {X -0.002,Y -406.773,Z 769.844,A 0.000,B 0.000,C 90.000,E1 187.992} C_DIS
LIN {X -0.051,Y -402.166,Z 769.829,A 0.000,B 0.000,C 90.000,E1 185.220} C_DIS
LIN {X 0.095,Y -398.453,Z 769.815,A 0.000,B 0.000,C 90.000,E1 182.751} C_DIS
LIN {X -0.027,Y -394.342,Z 769.798,A 0.000,B 0.000,C 90.000,E1 179.599} C_DIS
LIN {X -0.132,Y -391.565,Z 769.784,A 0.000,B 0.000,C 90.000,E1 177.135} C_DIS
LIN {X 0.050,Y -388.940,Z 769.768,A 0.000,B 0.000,C 90.000,E1 174.261} C_DIS
LIN {X -0.160,Y -386.670,Z 769.752,A 0.000,B 0.000,C 90.000,E1 171.432} C_DIS
LIN {X -0.118,Y -385.147,Z 769.740,A 0.000,B 0.000,C 90.000,E1 169.275} C_DIS
LIN {X -0.113,Y -383.793,Z 769.728,A 0.000,B 0.000,C 90.000,E1 167.117} C_DIS
LIN {X 0.020,Y -382.800,Z 769.716,A 0.000,B 0.000,C 90.000,E1 164.936} C_DIS
LIN {X -0.038,Y -381.961,Z 769.704,A 0.000,B 0.000,C 90.000,E1 162.779} C_DIS
LIN {X 0.018,Y -380.907,Z 769.684,A 0.000,B 0.000,C 90.000,E1 159.156} C_DIS
LIN {X 0.221,Y -380.629,Z 769.668,A 0.000,B 0.000,C 90.000,E1 156.230} C_DIS
LIN {X 0.099,Y -380.944,Z 769.656,A 0.000,B 0.000,C 90.000,E1 154.076} C_DIS
LIN {X -0.033,Y -381.742,Z 769.642,A 0.000,B 0.000,C 90.000,E1 151.563} C_DIS
LIN {X 0.058,Y -382.851,Z 769.632,A 0.000,B 0.000,C 90.000,E1 149.744} C_DIS
LIN {X 0.028,Y -384.656,Z 769.622,A 0.000,B 0.000,C 90.000,E1 147.946} C_DIS
LIN {X -0.211,Y -387.851,Z 769.608,A 0.000,B 0.000,C 90.000,E1 145.468} C_DIS
LIN {X 0.056,Y -389.827,Z 769.602,A 0.000,B 0.000,C 90.000,E1 144.356} C_DIS
LIN {X 0.029,Y -392.168,Z 769.596,A 0.000,B 0.000,C 90.000,E1 143.290} C_DIS
LIN {X 0.105,Y -393.027,Z 769.594,A 0.000,B 0.000,C 90.000,E1 142.924} C_DIS
LIN {X -0.033,Y -395.192,Z 769.590,A 0.000,B 0.000,C 90.000,E1 142.236} C_DIS
LIN {X -0.090,Y -397.975,Z 769.586,A 0.000,B 0.000,C 90.000,E1 141.537} C_DIS
LIN {X 0.186,Y -400.074,Z 769.584,A 0.000,B 0.000,C 90.000,E1 141.090} C_DIS
LIN {X 0.085,Y -400.886,Z 769.583,A 0.000,B 0.000,C 90.000,E1 140.928} C_DIS
LIN {X -0.148,Y -404.093,Z 769.580,A 0.000,B 0.000,C 90.000,E1 140.436} C_DIS
LIN {X 0.065,Y -408.288,Z 769.577,A 0.000,B 0.000,C 90.000,E1 139.828} C_DIS
LIN {X -0.148,Y -414.712,Z 769.573,A 0.000,B 0.000,C 90.000,E1 139.094} C_DIS
LIN {X 0.018,Y -433.223,Z 769.562,A 0.000,B 0.000,C 90.000,E1 137.106} C_DIS
LIN {X 0.180,Y -441.630,Z 769.557,A 0.000,B 0.000,C 90.000,E1 136.215} C_DIS
LIN {X -0.006,Y -449.786,Z 769.552,A 0.000,B 0.000,C 90.000,E1 135.364} C_DIS
LIN {X 0.173,Y -458.019,Z 769.547,A 0.000,B 0.000,C 90.000,E1 134.433} C_DIS
LIN {X -0.188,Y -464.697,Z 769.543,A 0.000,B 0.000,C 90.000,E1 133.704} C_DIS
LIN {X -0.211,Y -471.163,Z 769.538,A 0.000,B 0.000,C 90.000,E1 132.933} C_DIS
LIN {X -0.020,Y -477.290,Z 769.534,A 0.000,B 0.000,C 90.000,E1 132.162} C_DIS
LIN {X -0.059,Y -483.420,Z 769.530,A 0.000,B 0.000,C 90.000,E1 131.391} C_DIS
LIN {X -0.114,Y -488.026,Z 769.527,A 0.000,B 0.000,C 90.000,E1 130.782} C_DIS
LIN {X -0.136,Y -492.450,Z 769.523,A 0.000,B 0.000,C 90.000,E1 130.172} C_DIS
LIN {X 0.034,Y -497.604,Z 769.519,A 0.000,B 0.000,C 90.000,E1 129.402} C_DIS
LIN {X -0.012,Y -500.577,Z 769.516,A 0.000,B 0.000,C 90.000,E1 128.955} C_DIS
LIN {X -0.228,Y -504.383,Z 769.513,A 0.000,B 0.000,C 90.000,E1 128.382} C_DIS
LIN {X 0.264,Y -508.069,Z 769.510,A 0.000,B 0.000,C 90.000,E1 127.729} C_DIS
LIN {X -0.125,Y -512.348,Z 769.506,A 0.000,B 0.000,C 90.000,E1 127.030} C_DIS
LIN {X -0.050,Y -517.280,Z 769.501,A 0.000,B 0.000,C 90.000,E1 126.137} C_DIS
LIN {X 0.014,Y -522.729,Z 769.495,A 0.000,B 0.000,C 90.000,E1 125.105} C_DIS
LIN {X -0.076,Y -525.615,Z 769.492,A 0.000,B 0.000,C 90.000,E1 124.532} C_DIS
LIN {X -0.034,Y -529.563,Z 769.487,A 0.000,B 0.000,C 90.000,E1 123.658} C_DIS
LIN {X -0.100,Y -533.283,Z 769.482,A 0.000,B 0.000,C 90.000,E1 122.801} C_DIS
LIN {X -0.118,Y -537.453,Z 769.477,A 0.000,B 0.000,C 90.000,E1 121.799} C_DIS
LIN {X 0.056,Y -540.755,Z 769.472,A 0.000,B 0.000,C 90.000,E1 120.924} C_DIS
LIN {X -0.010,Y -543.802,Z 769.467,A 0.000,B 0.000,C 90.000,E1 120.079} C_DIS
LIN {X -0.020,Y -547.545,Z 769.461,A 0.000,B 0.000,C 90.000,E1 118.949} C_DIS
LIN {X -0.006,Y -550.246,Z 769.456,A 0.000,B 0.000,C 90.000,E1 118.103} C_DIS
LIN {X 0.036,Y -552.812,Z 769.451,A 0.000,B 0.000,C 90.000,E1 117.257} C_DIS
LIN {X 0.100,Y -555.050,Z 769.447,A 0.000,B 0.000,C 90.000,E1 116.411} C_DIS
LIN {X 0.016,Y -557.921,Z 769.439,A 0.000,B 0.000,C 90.000,E1 115.027} C_DIS
LIN {X 0.101,Y -558.827,Z 769.436,A 0.000,B 0.000,C 90.000,E1 114.463} C_DIS
LIN {X 0.087,Y -560.715,Z 769.428,A 0.000,B 0.000,C 90.000,E1 113.078} C_DIS
LIN {X -0.118,Y -562.550,Z 769.421,A 0.000,B 0.000,C 90.000,E1 111.716} C_DIS
LIN {X -0.170,Y -564.420,Z 769.411,A 0.000,B 0.000,C 90.000,E1 110.066} C_DIS
LIN {X -0.122,Y -565.567,Z 769.405,A 0.000,B 0.000,C 90.000,E1 108.960} C_DIS
LIN {X -0.095,Y -566.825,Z 769.398,A 0.000,B 0.000,C 90.000,E1 107.583} C_DIS
LIN {X -0.089,Y -568.526,Z 769.387,A 0.000,B 0.000,C 90.000,E1 105.662} C_DIS
LIN {X 0.021,Y -569.903,Z 769.378,A 0.000,B 0.000,C 90.000,E1 104.008} C_DIS
LIN {X -0.208,Y -571.682,Z 769.367,A 0.000,B 0.000,C 90.000,E1 102.119} C_DIS
LIN {X 0.123,Y -573.747,Z 769.355,A 0.000,B 0.000,C 90.000,E1 99.905} C_DIS
LIN {X -0.102,Y -574.882,Z 769.348,A 0.000,B 0.000,C 90.000,E1 98.568} C_DIS
LIN {X 0.179,Y -576.004,Z 769.340,A 0.000,B 0.000,C 90.000,E1 97.182} C_DIS
LIN {X -0.096,Y -576.977,Z 769.333,A 0.000,B 0.000,C 90.000,E1 95.853} C_DIS
LIN {X 0.012,Y -577.682,Z 769.326,A 0.000,B 0.000,C 90.000,E1 94.759} C_DIS
LIN {X -0.149,Y -578.769,Z 769.318,A 0.000,B 0.000,C 90.000,E1 93.151} C_DIS
LIN {X 0.260,Y -579.621,Z 769.308,A 0.000,B 0.000,C 90.000,E1 91.489} C_DIS
LIN {X 0.101,Y -580.427,Z 769.299,A 0.000,B 0.000,C 90.000,E1 89.885} C_DIS
LIN {X -0.213,Y -580.960,Z 769.292,A 0.000,B 0.000,C 90.000,E1 88.568} C_DIS
LIN {X 0.074,Y -581.406,Z 769.284,A 0.000,B 0.000,C 90.000,E1 87.192} C_DIS
LIN {X -0.006,Y -581.852,Z 769.276,A 0.000,B 0.000,C 90.000,E1 85.584} C_DIS
LIN {X -0.022,Y -582.158,Z 769.267,A 0.000,B 0.000,C 90.000,E1 83.970} C_DIS
LIN {X -0.031,Y -582.333,Z 769.258,A 0.000,B 0.000,C 90.000,E1 82.356} C_DIS
LIN {X 0.031,Y -582.387,Z 769.249,A 0.000,B 0.000,C 90.000,E1 80.735} C_DIS
LIN {X -0.281,Y -582.458,Z 769.243,A 0.000,B 0.000,C 90.000,E1 79.690} C_DIS
LIN {X -0.248,Y -582.368,Z 769.235,A 0.000,B 0.000,C 90.000,E1 78.342} C_DIS
LIN {X 0.022,Y -582.041,Z 769.226,A 0.000,B 0.000,C 90.000,E1 76.700} C_DIS
LIN {X 0.039,Y -581.645,Z 769.219,A 0.000,B 0.000,C 90.000,E1 75.353} C_DIS
LIN {X 0.004,Y -581.033,Z 769.210,A 0.000,B 0.000,C 90.000,E1 73.740} C_DIS
LIN {X -0.039,Y -580.364,Z 769.201,A 0.000,B 0.000,C 90.000,E1 72.127} C_DIS
LIN {X -0.121,Y -579.690,Z 769.193,A 0.000,B 0.000,C 90.000,E1 70.786} C_DIS
LIN {X -0.180,Y -578.534,Z 769.183,A 0.000,B 0.000,C 90.000,E1 68.901} C_DIS
LIN {X 0.069,Y -577.731,Z 769.177,A 0.000,B 0.000,C 90.000,E1 67.794} C_DIS
LIN {X 0.147,Y -576.617,Z 769.169,A 0.000,B 0.000,C 90.000,E1 66.433} C_DIS
LIN {X 0.062,Y -575.597,Z 769.163,A 0.000,B 0.000,C 90.000,E1 65.357} C_DIS
LIN {X -0.188,Y -574.150,Z 769.156,A 0.000,B 0.000,C 90.000,E1 64.024} C_DIS
LIN {X -0.205,Y -572.386,Z 769.148,A 0.000,B 0.000,C 90.000,E1 62.666} C_DIS
LIN {X -0.085,Y -570.669,Z 769.142,A 0.000,B 0.000,C 90.000,E1 61.563} C_DIS
LIN {X 0.182,Y -569.241,Z 769.137,A 0.000,B 0.000,C 90.000,E1 60.717} C_DIS
LIN {X -0.244,Y -567.157,Z 769.131,A 0.000,B 0.000,C 90.000,E1 59.665} C_DIS
LIN {X -0.027,Y -565.366,Z 769.127,A 0.000,B 0.000,C 90.000,E1 58.820} C_DIS
LIN {X -0.022,Y -563.345,Z 769.122,A 0.000,B 0.000,C 90.000,E1 57.995} C_DIS
LIN {X -0.243,Y -560.339,Z 769.116,A 0.000,B 0.000,C 90.000,E1 56.914} C_DIS
LIN {X -0.284,Y -557.883,Z 769.112,A 0.000,B 0.000,C 90.000,E1 56.087} C_DIS
LIN {X -0.116,Y -556.179,Z 769.108,A 0.000,B 0.000,C 90.000,E1 55.515} C_DIS
LIN {X -0.200,Y -553.333,Z 769.104,A 0.000,B 0.000,C 90.000,E1 54.689} C_DIS
LIN {X 0.005,Y -550.068,Z 769.099,A 0.000,B 0.000,C 90.000,E1 53.829} C_DIS
LIN {X -0.015,Y -547.070,Z 769.095,A 0.000,B 0.000,C 90.000,E1 53.130} C_DIS
LIN {X -0.070,Y -543.822,Z 769.091,A 0.000,B 0.000,C 90.000,E1 52.431} C_DIS
LIN {X 0.172,Y -540.283,Z 769.087,A 0.000,B 0.000,C 90.000,E1 51.698} C_DIS
LIN {X -0.212,Y -537.252,Z 769.084,A 0.000,B 0.000,C 90.000,E1 51.170} C_DIS
LIN {X 0.143,Y -533.953,Z 769.081,A 0.000,B 0.000,C 90.000,E1 50.561} C_DIS
LIN {X 0.131,Y -530.217,Z 769.078,A 0.000,B 0.000,C 90.000,E1 49.989} C_DIS
LIN {X -0.313,Y -526.151,Z 769.075,A 0.000,B 0.000,C 90.000,E1 49.461} C_DIS
LIN {X 0.105,Y -520.203,Z 769.071,A 0.000,B 0.000,C 90.000,E1 48.690} C_DIS
LIN {X 0.192,Y -516.359,Z 769.068,A 0.000,B 0.000,C 90.000,E1 48.243} C_DIS
LIN {X 0.009,Y -512.334,Z 769.066,A 0.000,B 0.000,C 90.000,E1 47.838} C_DIS
LIN {X -0.206,Y -506.548,Z 769.063,A 0.000,B 0.000,C 90.000,E1 47.310} C_DIS
LIN {X -0.102,Y -502.142,Z 769.061,A 0.000,B 0.000,C 90.000,E1 46.905} C_DIS
LIN {X 0.175,Y -496.012,Z 769.058,A 0.000,B 0.000,C 90.000,E1 46.377} C_DIS
LIN {X 0.110,Y -491.809,Z 769.056,A 0.000,B 0.000,C 90.000,E1 46.053} C_DIS
LIN {X 0.195,Y -485.409,Z 769.053,A 0.000,B 0.000,C 90.000,E1 45.567} C_DIS
LIN {X -0.202,Y -478.895,Z 769.051,A 0.000,B 0.000,C 90.000,E1 45.162} C_DIS
LIN {X 0.097,Y -466.059,Z 769.046,A 0.000,B 0.000,C 90.000,E1 44.271} C_DIS
LIN {X 0.223,Y -444.990,Z 769.038,A 0.000,B 0.000,C 90.000,E1 42.852} C_DIS
LIN {X -0.053,Y -422.789,Z 769.029,A 0.000,B 0.000,C 90.000,E1 41.310} C_DIS
LIN {X 0.258,Y -413.641,Z 769.025,A 0.000,B 0.000,C 90.000,E1 40.539} C_DIS
LIN {X 0.108,Y -408.611,Z 769.023,A 0.000,B 0.000,C 90.000,E1 40.092} C_DIS
LIN {X 0.076,Y -408.577,Z 769.023,A 0.000,B 0.000,C 90.000,E1 40.092} C_DIS
LIN {X -0.095,Y -405.941,Z 769.014,A 0.000,B 0.000,C 90.000,E1 38.543} C_DIS
LIN {X 0.141,Y -398.849,Z 768.995,A 0.000,B 0.000,C 90.000,E1 35.025} C_DIS
LIN {X 0.021,Y -398.735,Z 768.993,A 0.000,B 0.000,C 90.000,E1 34.692} C_DIS
LIN {X -0.061,Y -399.431,Z 768.975,A 0.000,B 0.000,C 90.000,E1 31.544} C_DIS
LIN {X 0.149,Y -400.777,Z 768.958,A 0.000,B 0.000,C 90.000,E1 28.359} C_DIS
LIN {X -0.061,Y -402.421,Z 768.942,A 0.000,B 0.000,C 90.000,E1 25.591} C_DIS
LIN {X 0.108,Y -403.537,Z 768.932,A 0.000,B 0.000,C 90.000,E1 23.823} C_DIS
LIN {X 0.136,Y -404.911,Z 768.923,A 0.000,B 0.000,C 90.000,E1 22.078} C_DIS
LIN {X 0.212,Y -408.362,Z 768.904,A 0.000,B 0.000,C 90.000,E1 18.598} C_DIS
LIN {X -0.072,Y -412.940,Z 768.884,A 0.000,B 0.000,C 90.000,E1 15.190} C_DIS
LIN {X 0.035,Y -416.062,Z 768.873,A 0.000,B 0.000,C 90.000,E1 13.119} C_DIS
LIN {X 0.035,Y -419.376,Z 768.862,A 0.000,B 0.000,C 90.000,E1 11.074} C_DIS
LIN {X 0.037,Y -422.193,Z 768.852,A 0.000,B 0.000,C 90.000,E1 9.378} C_DIS
LIN {X 0.038,Y -425.668,Z 768.841,A 0.000,B 0.000,C 90.000,E1 7.352} C_DIS
LIN {X 0.224,Y -430.290,Z 768.826,A 0.000,B 0.000,C 90.000,E1 4.645} C_DIS
LIN {X 0.038,Y -435.215,Z 768.811,A 0.000,B 0.000,C 90.000,E1 2.007} C_DIS
LIN {X 0.166,Y -439.576,Z 768.799,A 0.000,B 0.000,C 90.000,E1 359.771} C_DIS
LIN {X 0.135,Y -444.290,Z 768.786,A 0.000,B 0.000,C 90.000,E1 357.478} C_DIS
LIN {X -0.022,Y -450.142,Z 768.772,A 0.000,B 0.000,C 90.000,E1 354.894} C_DIS
LIN {X -0.039,Y -453.937,Z 768.763,A 0.000,B 0.000,C 90.000,E1 353.280} C_DIS
LIN {X -0.146,Y -456.929,Z 768.756,A 0.000,B 0.000,C 90.000,E1 352.008} C_DIS
LIN {X 0.025,Y -460.504,Z 768.747,A 0.000,B 0.000,C 90.000,E1 350.387} C_DIS
LIN {X -0.117,Y -463.848,Z 768.738,A 0.000,B 0.000,C 90.000,E1 348.814} C_DIS
LIN {X -0.106,Y -469.310,Z 768.724,A 0.000,B 0.000,C 90.000,E1 346.284} C_DIS
LIN {X -0.022,Y -471.225,Z 768.720,A 0.000,B 0.000,C 90.000,E1 345.644} C_DIS
LIN {X -0.006,Y -473.069,Z 768.718,A 0.000,B 0.000,C 90.000,E1 345.172} C_DIS
LIN {X -0.060,Y -474.710,Z 768.716,A 0.000,B 0.000,C 90.000,E1 344.866} C_DIS
LIN {X -0.035,Y -478.113,Z 768.713,A 0.000,B 0.000,C 90.000,E1 344.338} C_DIS
LIN {X -0.067,Y -480.701,Z 768.711,A 0.000,B 0.000,C 90.000,E1 344.031} C_DIS
LIN {X -0.161,Y -487.585,Z 768.708,A 0.000,B 0.000,C 90.000,E1 343.378} C_DIS
LIN {X -0.053,Y -494.480,Z 768.705,A 0.000,B 0.000,C 90.000,E1 342.834} C_DIS
LIN {X 0.013,Y -516.312,Z 768.696,A 0.000,B 0.000,C 90.000,E1 341.329} C_DIS
LIN {X 0.146,Y -537.096,Z 768.689,A 0.000,B 0.000,C 90.000,E1 340.007} C_DIS
LIN {X 0.222,Y -541.726,Z 768.687,A 0.000,B 0.000,C 90.000,E1 339.699} C_DIS
LIN {X -0.129,Y -547.704,Z 768.685,A 0.000,B 0.000,C 90.000,E1 339.316} C_DIS
LIN {X 0.029,Y -553.411,Z 768.683,A 0.000,B 0.000,C 90.000,E1 338.847} C_DIS
LIN {X 0.055,Y -558.881,Z 768.680,A 0.000,B 0.000,C 90.000,E1 338.358} C_DIS
LIN {X 0.038,Y -564.100,Z 768.677,A 0.000,B 0.000,C 90.000,E1 337.847} C_DIS
LIN {X 0.073,Y -570.339,Z 768.673,A 0.000,B 0.000,C 90.000,E1 337.177} C_DIS
LIN {X -0.186,Y -573.977,Z 768.671,A 0.000,B 0.000,C 90.000,E1 336.794} C_DIS
LIN {X 0.327,Y -581.759,Z 768.666,A 0.000,B 0.000,C 90.000,E1 335.793} C_DIS
LIN {X -0.121,Y -588.931,Z 768.661,A 0.000,B 0.000,C 90.000,E1 334.897} C_DIS
LIN {X 0.050,Y -595.632,Z 768.655,A 0.000,B 0.000,C 90.000,E1 333.948} C_DIS
LIN {X -0.161,Y -600.306,Z 768.652,A 0.000,B 0.000,C 90.000,E1 333.307} C_DIS
LIN {X 0.171,Y -605.622,Z 768.647,A 0.000,B 0.000,C 90.000,E1 332.487} C_DIS
LIN {X 0.264,Y -612.345,Z 768.641,A 0.000,B 0.000,C 90.000,E1 331.435} C_DIS
LIN {X 0.160,Y -617.899,Z 768.636,A 0.000,B 0.000,C 90.000,E1 330.539} C_DIS
LIN {X -0.120,Y -624.077,Z 768.631,A 0.000,B 0.000,C 90.000,E1 329.537} C_DIS
LIN {X -0.320,Y -629.798,Z 768.625,A 0.000,B 0.000,C 90.000,E1 328.535} C_DIS
LIN {X -0.107,Y -635.259,Z 768.619,A 0.000,B 0.000,C 90.000,E1 327.502} C_DIS
LIN {X -0.201,Y -639.027,Z 768.615,A 0.000,B 0.000,C 90.000,E1 326.755} C_DIS
LIN {X 0.141,Y -643.731,Z 768.610,A 0.000,B 0.000,C 90.000,E1 325.722} C_DIS
LIN {X 0.118,Y -647.121,Z 768.606,A 0.000,B 0.000,C 90.000,E1 324.975} C_DIS
LIN {X -0.058,Y -652.371,Z 768.599,A 0.000,B 0.000,C 90.000,E1 323.749} C_DIS
LIN {X -0.078,Y -656.273,Z 768.593,A 0.000,B 0.000,C 90.000,E1 322.763} C_DIS
LIN {X -0.103,Y -660.816,Z 768.586,A 0.000,B 0.000,C 90.000,E1 321.537} C_DIS
LIN {X -0.086,Y -665.785,Z 768.578,A 0.000,B 0.000,C 90.000,E1 320.070} C_DIS
LIN {X -0.054,Y -669.683,Z 768.571,A 0.000,B 0.000,C 90.000,E1 318.852} C_DIS
LIN {X 0.042,Y -673.235,Z 768.565,A 0.000,B 0.000,C 90.000,E1 317.634} C_DIS
LIN {X -0.307,Y -676.321,Z 768.558,A 0.000,B 0.000,C 90.000,E1 316.458} C_DIS
LIN {X -0.176,Y -678.611,Z 768.553,A 0.000,B 0.000,C 90.000,E1 315.486} C_DIS
LIN {X -0.055,Y -680.159,Z 768.549,A 0.000,B 0.000,C 90.000,E1 314.757} C_DIS
LIN {X 0.178,Y -682.563,Z 768.542,A 0.000,B 0.000,C 90.000,E1 313.542} C_DIS
LIN {X -0.026,Y -684.780,Z 768.535,A 0.000,B 0.000,C 90.000,E1 312.366} C_DIS
LIN {X 0.314,Y -686.808,Z 768.529,A 0.000,B 0.000,C 90.000,E1 311.148} C_DIS
LIN {X 0.100,Y -688.179,Z 768.523,A 0.000,B 0.000,C 90.000,E1 310.216} C_DIS
LIN {X -0.330,Y -689.902,Z 768.516,A 0.000,B 0.000,C 90.000,E1 308.830} C_DIS
LIN {X 0.192,Y -691.260,Z 768.509,A 0.000,B 0.000,C 90.000,E1 307.604} C_DIS
LIN {X -0.230,Y -692.355,Z 768.503,A 0.000,B 0.000,C 90.000,E1 306.457} C_DIS
LIN {X 0.326,Y -693.399,Z 768.496,A 0.000,B 0.000,C 90.000,E1 305.231} C_DIS
LIN {X 0.101,Y -694.316,Z 768.489,A 0.000,B 0.000,C 90.000,E1 304.072} C_DIS
LIN {X -0.073,Y -695.375,Z 768.482,A 0.000,B 0.000,C 90.000,E1 302.673} C_DIS
LIN {X -0.027,Y -696.483,Z 768.474,A 0.000,B 0.000,C 90.000,E1 301.258} C_DIS
LIN {X 0.033,Y -697.259,Z 768.467,A 0.000,B 0.000,C 90.000,E1 300.079} C_DIS
LIN {X 0.116,Y -697.727,Z 768.461,A 0.000,B 0.000,C 90.000,E1 298.899} C_DIS
LIN {X -0.060,Y -698.112,Z 768.455,A 0.000,B 0.000,C 90.000,E1 297.975} C_DIS
LIN {X -0.384,Y -698.799,Z 768.446,A 0.000,B 0.000,C 90.000,E1 296.360} C_DIS
LIN {X 0.021,Y -699.481,Z 768.440,A 0.000,B 0.000,C 90.000,E1 295.155} C_DIS
LIN {X -0.079,Y -699.676,Z 768.437,A 0.000,B 0.000,C 90.000,E1 294.695} C_DIS
LIN {X 0.166,Y -699.361,Z 768.435,A 0.000,B 0.000,C 90.000,E1 294.207} C_DIS
LIN {X -0.206,Y -698.999,Z 768.433,A 0.000,B 0.000,C 90.000,E1 294.003} C_DIS
LIN {X 0.040,Y -697.453,Z 768.431,A 0.000,B 0.000,C 90.000,E1 293.515} C_DIS
LIN {X 0.299,Y -696.243,Z 768.429,A 0.000,B 0.000,C 90.000,E1 293.259} C_DIS
LIN {X 0.153,Y -695.149,Z 768.429,A 0.000,B 0.000,C 90.000,E1 293.153} C_DIS
LIN {X 0.089,Y -689.826,Z 768.426,A 0.000,B 0.000,C 90.000,E1 292.717} C_DIS
LIN {X -0.308,Y -687.922,Z 768.426,A 0.000,B 0.000,C 90.000,E1 292.642} C_DIS
LIN {X -0.213,Y -683.194,Z 768.425,A 0.000,B 0.000,C 90.000,E1 292.461} C_DIS
LIN {X 0.251,Y -675.039,Z 768.424,A 0.000,B 0.000,C 90.000,E1 292.206} C_DIS
LIN {X 0.033,Y -665.757,Z 768.423,A 0.000,B 0.000,C 90.000,E1 292.078} C_DIS
LIN {X -0.146,Y -654.749,Z 768.422,A 0.000,B 0.000,C 90.000,E1 291.950} C_DIS
LIN {X 0.025,Y -644.682,Z 768.421,A 0.000,B 0.000,C 90.000,E1 291.770} C_DIS
LIN {X -0.092,Y -635.262,Z 768.420,A 0.000,B 0.000,C 90.000,E1 291.589} C_DIS
LIN {X -0.086,Y -614.171,Z 768.417,A 0.000,B 0.000,C 90.000,E1 291.099} C_DIS
LIN {X -0.212,Y -596.926,Z 768.415,A 0.000,B 0.000,C 90.000,E1 290.663} C_DIS
LIN {X -0.323,Y -575.941,Z 768.411,A 0.000,B 0.000,C 90.000,E1 290.066} C_DIS
LIN {X -0.287,Y -565.716,Z 768.410,A 0.000,B 0.000,C 90.000,E1 289.758} C_DIS
LIN {X -0.006,Y -559.067,Z 768.408,A 0.000,B 0.000,C 90.000,E1 289.450} C_DIS
LIN {X 0.060,Y -556.657,Z 768.407,A 0.000,B 0.000,C 90.000,E1 289.214} C_DIS
LIN {X 0.021,Y -556.625,Z 768.407,A 0.000,B 0.000,C 90.000,E1 289.214} C_DIS
LIN {X 0.195,Y -555.776,Z 768.406,A 0.000,B 0.000,C 90.000,E1 288.960} C_DIS
LIN {X 0.024,Y -555.111,Z 768.402,A 0.000,B 0.000,C 90.000,E1 288.417} C_DIS
LIN {X -0.136,Y -554.494,Z 768.395,A 0.000,B 0.000,C 90.000,E1 287.040} C_DIS
LIN {X -0.102,Y -553.351,Z 768.379,A 0.000,B 0.000,C 90.000,E1 284.245} C_DIS
LIN {X 0.096,Y -552.834,Z 768.371,A 0.000,B 0.000,C 90.000,E1 282.827} C_DIS
LIN {X 0.161,Y -552.383,Z 768.364,A 0.000,B 0.000,C 90.000,E1 281.422} C_DIS
LIN {X -0.191,Y -551.681,Z 768.353,A 0.000,B 0.000,C 90.000,E1 279.500} C_DIS
LIN {X -0.102,Y -551.104,Z 768.342,A 0.000,B 0.000,C 90.000,E1 277.530} C_DIS
LIN {X -0.248,Y -550.412,Z 768.334,A 0.000,B 0.000,C 90.000,E1 276.144} C_DIS
LIN {X -0.006,Y -549.883,Z 768.329,A 0.000,B 0.000,C 90.000,E1 275.277} C_DIS
LIN {X -0.143,Y -548.599,Z 768.318,A 0.000,B 0.000,C 90.000,E1 273.326} C_DIS
LIN {X -0.266,Y -547.360,Z 768.306,A 0.000,B 0.000,C 90.000,E1 271.088} C_DIS
LIN {X 0.005,Y -546.273,Z 768.297,A 0.000,B 0.000,C 90.000,E1 269.370} C_DIS
LIN {X -0.246,Y -544.905,Z 768.286,A 0.000,B 0.000,C 90.000,E1 267.421} C_DIS
LIN {X 0.012,Y -543.856,Z 768.276,A 0.000,B 0.000,C 90.000,E1 265.698} C_DIS
LIN {X 0.237,Y -542.791,Z 768.267,A 0.000,B 0.000,C 90.000,E1 263.976} C_DIS
LIN {X -0.066,Y -541.695,Z 768.259,A 0.000,B 0.000,C 90.000,E1 262.591} C_DIS
LIN {X -0.248,Y -540.029,Z 768.248,A 0.000,B 0.000,C 90.000,E1 260.622} C_DIS
LIN {X 0.038,Y -539.039,Z 768.241,A 0.000,B 0.000,C 90.000,E1 259.454} C_DIS
LIN {X -0.078,Y -537.641,Z 768.232,A 0.000,B 0.000,C 90.000,E1 257.757} C_DIS
LIN {X -0.105,Y -536.075,Z 768.222,A 0.000,B 0.000,C 90.000,E1 256.047} C_DIS
LIN {X 0.017,Y -533.888,Z 768.211,A 0.000,B 0.000,C 90.000,E1 254.031} C_DIS
LIN {X -0.262,Y -531.304,Z 768.199,A 0.000,B 0.000,C 90.000,E1 251.764} C_DIS
LIN {X 0.130,Y -530.265,Z 768.194,A 0.000,B 0.000,C 90.000,E1 250.859} C_DIS
LIN {X 0.062,Y -527.838,Z 768.184,A 0.000,B 0.000,C 90.000,E1 249.135} C_DIS
LIN {X 0.266,Y -525.783,Z 768.176,A 0.000,B 0.000,C 90.000,E1 247.667} C_DIS
LIN {X 0.140,Y -523.582,Z 768.168,A 0.000,B 0.000,C 90.000,E1 246.230} C_DIS
LIN {X -0.178,Y -521.746,Z 768.162,A 0.000,B 0.000,C 90.000,E1 245.101} C_DIS
LIN {X -0.159,Y -519.374,Z 768.154,A 0.000,B 0.000,C 90.000,E1 243.640} C_DIS
LIN {X 0.016,Y -517.893,Z 768.149,A 0.000,B 0.000,C 90.000,E1 242.743} C_DIS
LIN {X 0.077,Y -515.755,Z 768.142,A 0.000,B 0.000,C 90.000,E1 241.563} C_DIS
LIN {X -0.236,Y -512.908,Z 768.134,A 0.000,B 0.000,C 90.000,E1 240.127} C_DIS
LIN {X 0.088,Y -510.043,Z 768.126,A 0.000,B 0.000,C 90.000,E1 238.614} C_DIS
LIN {X 0.182,Y -507.158,Z 768.117,A 0.000,B 0.000,C 90.000,E1 237.120} C_DIS
LIN {X -0.092,Y -504.625,Z 768.111,A 0.000,B 0.000,C 90.000,E1 235.960} C_DIS
LIN {X -0.236,Y -501.125,Z 768.103,A 0.000,B 0.000,C 90.000,E1 234.482} C_DIS
LIN {X -0.016,Y -498.198,Z 768.096,A 0.000,B 0.000,C 90.000,E1 233.256} C_DIS
LIN {X -0.259,Y -492.853,Z 768.084,A 0.000,B 0.000,C 90.000,E1 231.170} C_DIS
LIN {X -0.030,Y -487.796,Z 768.072,A 0.000,B 0.000,C 90.000,E1 229.013} C_DIS
LIN {X 0.200,Y -483.671,Z 768.062,A 0.000,B 0.000,C 90.000,E1 227.148} C_DIS
LIN {X -0.140,Y -480.380,Z 768.054,A 0.000,B 0.000,C 90.000,E1 225.648} C_DIS
LIN {X -0.204,Y -477.077,Z 768.045,A 0.000,B 0.000,C 90.000,E1 224.109} C_DIS
LIN {X 0.007,Y -473.696,Z 768.036,A 0.000,B 0.000,C 90.000,E1 222.528} C_DIS
LIN {X 0.058,Y -470.959,Z 768.029,A 0.000,B 0.000,C 90.000,E1 221.272} C_DIS
LIN {X -0.122,Y -467.598,Z 768.021,A 0.000,B 0.000,C 90.000,E1 219.725} C_DIS
LIN {X 0.298,Y -464.232,Z 768.012,A 0.000,B 0.000,C 90.000,E1 218.096} C_DIS
LIN {X -0.152,Y -459.590,Z 768.000,A 0.000,B 0.000,C 90.000,E1 215.931} C_DIS
LIN {X -0.081,Y -456.330,Z 767.991,A 0.000,B 0.000,C 90.000,E1 214.326} C_DIS
LIN {X 0.056,Y -453.121,Z 767.982,A 0.000,B 0.000,C 90.000,E1 212.704} C_DIS
LIN {X -0.001,Y -448.148,Z 767.967,A 0.000,B 0.000,C 90.000,E1 210.129} C_DIS
LIN {X -0.013,Y -444.464,Z 767.957,A 0.000,B 0.000,C 90.000,E1 208.180} C_DIS
LIN {X 0.001,Y -442.016,Z 767.949,A 0.000,B 0.000,C 90.000,E1 206.873} C_DIS
LIN {X 0.039,Y -438.365,Z 767.938,A 0.000,B 0.000,C 90.000,E1 204.899} C_DIS
LIN {X 0.032,Y -433.984,Z 767.926,A 0.000,B 0.000,C 90.000,E1 202.589} C_DIS
LIN {X 0.072,Y -432.077,Z 767.920,A 0.000,B 0.000,C 90.000,E1 201.589} C_DIS
LIN {X -0.047,Y -428.880,Z 767.911,A 0.000,B 0.000,C 90.000,E1 199.939} C_DIS
LIN {X 0.174,Y -425.713,Z 767.901,A 0.000,B 0.000,C 90.000,E1 198.236} C_DIS
LIN {X 0.070,Y -422.520,Z 767.892,A 0.000,B 0.000,C 90.000,E1 196.567} C_DIS
LIN {X 0.075,Y -418.480,Z 767.881,A 0.000,B 0.000,C 90.000,E1 194.537} C_DIS
LIN {X -0.093,Y -414.122,Z 767.868,A 0.000,B 0.000,C 90.000,E1 192.175} C_DIS
LIN {X -0.158,Y -409.890,Z 767.854,A 0.000,B 0.000,C 90.000,E1 189.782} C_DIS
LIN {X -0.102,Y -406.948,Z 767.845,A 0.000,B 0.000,C 90.000,E1 188.049} C_DIS
LIN {X -0.147,Y -402.332,Z 767.829,A 0.000,B 0.000,C 90.000,E1 185.277} C_DIS
LIN {X 0.004,Y -398.639,Z 767.816,A 0.000,B 0.000,C 90.000,E1 182.808} C_DIS
LIN {X -0.111,Y -394.504,Z 767.798,A 0.000,B 0.000,C 90.000,E1 179.656} C_DIS
LIN {X 0.181,Y -391.716,Z 767.784,A 0.000,B 0.000,C 90.000,E1 177.135} C_DIS
LIN {X -0.022,Y -389.072,Z 767.768,A 0.000,B 0.000,C 90.000,E1 174.318} C_DIS
LIN {X 0.159,Y -386.859,Z 767.753,A 0.000,B 0.000,C 90.000,E1 171.432} C_DIS
LIN {X 0.135,Y -385.179,Z 767.739,A 0.000,B 0.000,C 90.000,E1 168.926} C_DIS
LIN {X 0.135,Y -383.895,Z 767.727,A 0.000,B 0.000,C 90.000,E1 166.769} C_DIS
LIN {X -0.007,Y -382.940,Z 767.715,A 0.000,B 0.000,C 90.000,E1 164.629} C_DIS
LIN {X -0.167,Y -382.076,Z 767.703,A 0.000,B 0.000,C 90.000,E1 162.489} C_DIS
LIN {X -0.139,Y -381.611,Z 767.695,A 0.000,B 0.000,C 90.000,E1 161.040} C_DIS
LIN {X 0.157,Y -381.072,Z 767.681,A 0.000,B 0.000,C 90.000,E1 158.465} C_DIS
LIN {X 0.020,Y -381.045,Z 767.662,A 0.000,B 0.000,C 90.000,E1 155.229} C_DIS
LIN {X -0.052,Y -382.536,Z 767.636,A 0.000,B 0.000,C 90.000,E1 150.539} C_DIS
LIN {X 0.086,Y -383.693,Z 767.628,A 0.000,B 0.000,C 90.000,E1 149.076} C_DIS
LIN {X -0.021,Y -386.842,Z 767.612,A 0.000,B 0.000,C 90.000,E1 146.215} C_DIS
LIN {X 0.016,Y -388.370,Z 767.606,A 0.000,B 0.000,C 90.000,E1 145.135} C_DIS
LIN {X 0.036,Y -391.015,Z 767.598,A 0.000,B 0.000,C 90.000,E1 143.703} C_DIS
LIN {X -0.052,Y -392.615,Z 767.594,A 0.000,B 0.000,C 90.000,E1 143.004} C_DIS
LIN {X -0.004,Y -395.204,Z 767.590,A 0.000,B 0.000,C 90.000,E1 142.110} C_DIS
LIN {X -0.019,Y -397.191,Z 767.587,A 0.000,B 0.000,C 90.000,E1 141.582} C_DIS
LIN {X -0.061,Y -400.429,Z 767.583,A 0.000,B 0.000,C 90.000,E1 140.884} C_DIS
LIN {X -0.043,Y -403.540,Z 767.580,A 0.000,B 0.000,C 90.000,E1 140.356} C_DIS
LIN {X 0.169,Y -407.643,Z 767.577,A 0.000,B 0.000,C 90.000,E1 139.747} C_DIS
LIN {X -0.075,Y -414.052,Z 767.572,A 0.000,B 0.000,C 90.000,E1 139.013} C_DIS
LIN {X -0.010,Y -429.958,Z 767.563,A 0.000,B 0.000,C 90.000,E1 137.310} C_DIS
LIN {X 0.008,Y -439.848,Z 767.557,A 0.000,B 0.000,C 90.000,E1 136.296} C_DIS
LIN {X -0.032,Y -448.353,Z 767.552,A 0.000,B 0.000,C 90.000,E1 135.405} C_DIS
LIN {X -0.015,Y -456.545,Z 767.547,A 0.000,B 0.000,C 90.000,E1 134.514} C_DIS
LIN {X 0.021,Y -464.703,Z 767.542,A 0.000,B 0.000,C 90.000,E1 133.581} C_DIS
LIN {X -0.104,Y -473.699,Z 767.536,A 0.000,B 0.000,C 90.000,E1 132.528} C_DIS
LIN {X -0.024,Y -481.105,Z 767.531,A 0.000,B 0.000,C 90.000,E1 131.595} C_DIS
LIN {X 0.139,Y -486.923,Z 767.527,A 0.000,B 0.000,C 90.000,E1 130.825} C_DIS
LIN {X -0.132,Y -492.556,Z 767.523,A 0.000,B 0.000,C 90.000,E1 130.092} C_DIS
LIN {X -0.124,Y -496.782,Z 767.519,A 0.000,B 0.000,C 90.000,E1 129.483} C_DIS
LIN {X 0.181,Y -502.749,Z 767.514,A 0.000,B 0.000,C 90.000,E1 128.543} C_DIS
LIN {X 0.055,Y -507.467,Z 767.510,A 0.000,B 0.000,C 90.000,E1 127.810} C_DIS
LIN {X -0.228,Y -512.645,Z 767.505,A 0.000,B 0.000,C 90.000,E1 126.950} C_DIS
LIN {X 0.265,Y -517.571,Z 767.500,A 0.000,B 0.000,C 90.000,E1 126.011} C_DIS
LIN {X 0.087,Y -522.297,Z 767.495,A 0.000,B 0.000,C 90.000,E1 125.152} C_DIS
LIN {X -0.306,Y -525.227,Z 767.492,A 0.000,B 0.000,C 90.000,E1 124.612} C_DIS
LIN {X 0.231,Y -529.109,Z 767.487,A 0.000,B 0.000,C 90.000,E1 123.706} C_DIS
LIN {X -0.130,Y -532.838,Z 767.483,A 0.000,B 0.000,C 90.000,E1 122.880} C_DIS
LIN {X -0.012,Y -537.632,Z 767.476,A 0.000,B 0.000,C 90.000,E1 121.720} C_DIS
LIN {X -0.116,Y -540.931,Z 767.471,A 0.000,B 0.000,C 90.000,E1 120.875} C_DIS
LIN {X -0.165,Y -544.913,Z 767.465,A 0.000,B 0.000,C 90.000,E1 119.745} C_DIS
LIN {X -0.163,Y -548.636,Z 767.459,A 0.000,B 0.000,C 90.000,E1 118.615} C_DIS
LIN {X 0.114,Y -552.148,Z 767.453,A 0.000,B 0.000,C 90.000,E1 117.462} C_DIS
LIN {X 0.177,Y -554.469,Z 767.448,A 0.000,B 0.000,C 90.000,E1 116.616} C_DIS
LIN {X -0.046,Y -555.178,Z 767.446,A 0.000,B 0.000,C 90.000,E1 116.360} C_DIS
LIN {X 0.113,Y -558.072,Z 767.439,A 0.000,B 0.000,C 90.000,E1 114.951} C_DIS
LIN {X -0.013,Y -559.383,Z 767.434,A 0.000,B 0.000,C 90.000,E1 114.131} C_DIS
LIN {X 0.066,Y -561.648,Z 767.425,A 0.000,B 0.000,C 90.000,E1 112.461} C_DIS
LIN {X -0.030,Y -562.734,Z 767.420,A 0.000,B 0.000,C 90.000,E1 111.642} C_DIS
LIN {X -0.087,Y -564.636,Z 767.411,A 0.000,B 0.000,C 90.000,E1 109.993} C_DIS
LIN {X -0.226,Y -565.802,Z 767.405,A 0.000,B 0.000,C 90.000,E1 108.906} C_DIS
LIN {X -0.020,Y -567.106,Z 767.397,A 0.000,B 0.000,C 90.000,E1 107.511} C_DIS
LIN {X -0.172,Y -568.815,Z 767.387,A 0.000,B 0.000,C 90.000,E1 105.607} C_DIS
LIN {X -0.236,Y -570.011,Z 767.379,A 0.000,B 0.000,C 90.000,E1 104.245} C_DIS
LIN {X -0.269,Y -572.055,Z 767.367,A 0.000,B 0.000,C 90.000,E1 102.063} C_DIS
LIN {X -0.123,Y -573.861,Z 767.356,A 0.000,B 0.000,C 90.000,E1 100.141} C_DIS
LIN {X 0.114,Y -574.837,Z 767.350,A 0.000,B 0.000,C 90.000,E1 99.029} C_DIS
LIN {X 0.021,Y -576.208,Z 767.341,A 0.000,B 0.000,C 90.000,E1 97.409} C_DIS
LIN {X -0.115,Y -577.407,Z 767.332,A 0.000,B 0.000,C 90.000,E1 95.796} C_DIS
LIN {X -0.274,Y -578.461,Z 767.323,A 0.000,B 0.000,C 90.000,E1 94.188} C_DIS
LIN {X 0.007,Y -579.359,Z 767.316,A 0.000,B 0.000,C 90.000,E1 92.808} C_DIS
LIN {X -0.146,Y -580.216,Z 767.307,A 0.000,B 0.000,C 90.000,E1 91.203} C_DIS
LIN {X 0.289,Y -581.019,Z 767.298,A 0.000,B 0.000,C 90.000,E1 89.542} C_DIS
LIN {X 0.173,Y -581.609,Z 767.289,A 0.000,B 0.000,C 90.000,E1 87.936} C_DIS
LIN {X -0.101,Y -582.013,Z 767.281,A 0.000,B 0.000,C 90.000,E1 86.617} C_DIS
LIN {X -0.164,Y -582.420,Z 767.272,A 0.000,B 0.000,C 90.000,E1 85.008} C_DIS
LIN {X 0.188,Y -582.646,Z 767.265,A 0.000,B 0.000,C 90.000,E1 83.628} C_DIS
LIN {X 0.256,Y -582.792,Z 767.256,A 0.000,B 0.000,C 90.000,E1 82.008} C_DIS
LIN {X -0.139,Y -582.843,Z 767.250,A 0.000,B 0.000,C 90.000,E1 80.971} C_DIS
LIN {X -0.214,Y -582.864,Z 767.242,A 0.000,B 0.000,C 90.000,E1 79.634} C_DIS
LIN {X -0.177,Y -582.739,Z 767.235,A 0.000,B 0.000,C 90.000,E1 78.285} C_DIS
LIN {X -0.236,Y -582.284,Z 767.224,A 0.000,B 0.000,C 90.000,E1 76.408} C_DIS
LIN {X -0.070,Y -581.862,Z 767.217,A 0.000,B 0.000,C 90.000,E1 75.046} C_DIS
LIN {X -0.089,Y -581.220,Z 767.208,A 0.000,B 0.000,C 90.000,E1 73.433} C_DIS
LIN {X 0.221,Y -580.624,Z 767.201,A 0.000,B 0.000,C 90.000,E1 72.054} C_DIS
LIN {X -0.040,Y -579.923,Z 767.193,A 0.000,B 0.000,C 90.000,E1 70.732} C_DIS
LIN {X 0.261,Y -578.866,Z 767.184,A 0.000,B 0.000,C 90.000,E1 69.082} C_DIS
LIN {X -0.019,Y -578.108,Z 767.178,A 0.000,B 0.000,C 90.000,E1 68.028} C_DIS
LIN {X 0.075,Y -576.970,Z 767.170,A 0.000,B 0.000,C 90.000,E1 66.666} C_DIS
LIN {X -0.236,Y -575.971,Z 767.164,A 0.000,B 0.000,C 90.000,E1 65.613} C_DIS
LIN {X 0.132,Y -574.172,Z 767.155,A 0.000,B 0.000,C 90.000,E1 63.948} C_DIS
LIN {X 0.017,Y -572.757,Z 767.149,A 0.000,B 0.000,C 90.000,E1 62.871} C_DIS
LIN {X 0.139,Y -571.087,Z 767.143,A 0.000,B 0.000,C 90.000,E1 61.769} C_DIS
LIN {X 0.234,Y -569.142,Z 767.137,A 0.000,B 0.000,C 90.000,E1 60.667} C_DIS
LIN {X 0.089,Y -566.983,Z 767.131,A 0.000,B 0.000,C 90.000,E1 59.587} C_DIS
LIN {X -0.180,Y -565.145,Z 767.127,A 0.000,B 0.000,C 90.000,E1 58.791} C_DIS
LIN {X 0.009,Y -563.073,Z 767.122,A 0.000,B 0.000,C 90.000,E1 57.946} C_DIS
LIN {X -0.008,Y -560.801,Z 767.117,A 0.000,B 0.000,C 90.000,E1 57.120} C_DIS
LIN {X 0.041,Y -557.469,Z 767.111,A 0.000,B 0.000,C 90.000,E1 56.008} C_DIS
LIN {X -0.108,Y -555.751,Z 767.108,A 0.000,B 0.000,C 90.000,E1 55.468} C_DIS
LIN {X 0.118,Y -552.799,Z 767.104,A 0.000,B 0.000,C 90.000,E1 54.609} C_DIS
LIN {X -0.008,Y -549.450,Z 767.099,A 0.000,B 0.000,C 90.000,E1 53.783} C_DIS
LIN {X 0.292,Y -546.381,Z 767.095,A 0.000,B 0.000,C 90.000,E1 53.050} C_DIS
LIN {X -0.200,Y -543.039,Z 767.091,A 0.000,B 0.000,C 90.000,E1 52.396} C_DIS
LIN {X -0.138,Y -540.189,Z 767.088,A 0.000,B 0.000,C 90.000,E1 51.823} C_DIS
LIN {X -0.099,Y -537.110,Z 767.085,A 0.000,B 0.000,C 90.000,E1 51.251} C_DIS
LIN {X 0.252,Y -533.749,Z 767.082,A 0.000,B 0.000,C 90.000,E1 50.642} C_DIS
LIN {X -0.327,Y -528.937,Z 767.078,A 0.000,B 0.000,C 90.000,E1 49.989} C_DIS
LIN {X -0.169,Y -525.878,Z 767.075,A 0.000,B 0.000,C 90.000,E1 49.542} C_DIS
LIN {X 0.241,Y -519.883,Z 767.071,A 0.000,B 0.000,C 90.000,E1 48.771} C_DIS
LIN {X -0.062,Y -515.964,Z 767.069,A 0.000,B 0.000,C 90.000,E1 48.366} C_DIS
LIN {X 0.123,Y -511.830,Z 767.066,A 0.000,B 0.000,C 90.000,E1 47.919} C_DIS
LIN {X -0.011,Y -506.110,Z 767.063,A 0.000,B 0.000,C 90.000,E1 47.391} C_DIS
LIN {X 0.078,Y -500.086,Z 767.060,A 0.000,B 0.000,C 90.000,E1 46.863} C_DIS
LIN {X 0.009,Y -495.498,Z 767.058,A 0.000,B 0.000,C 90.000,E1 46.500} C_DIS
LIN {X 0.098,Y -486.397,Z 767.055,A 0.000,B 0.000,C 90.000,E1 45.810} C_DIS
LIN {X -0.036,Y -478.631,Z 767.052,A 0.000,B 0.000,C 90.000,E1 45.283} C_DIS
LIN {X -0.234,Y -464.209,Z 767.046,A 0.000,B 0.000,C 90.000,E1 44.352} C_DIS
LIN {X -0.236,Y -441.674,Z 767.038,A 0.000,B 0.000,C 90.000,E1 42.852} C_DIS
LIN {X -0.151,Y -419.382,Z 767.029,A 0.000,B 0.000,C 90.000,E1 41.229} C_DIS
LIN {X 0.158,Y -413.454,Z 767.026,A 0.000,B 0.000,C 90.000,E1 40.701} C_DIS
LIN {X 0.102,Y -408.983,Z 767.024,A 0.000,B 0.000,C 90.000,E1 40.297} C_DIS
LIN {X 0.070,Y -408.945,Z 767.024,A 0.000,B 0.000,C 90.000,E1 40.297} C_DIS
LIN {X -0.163,Y -405.768,Z 767.014,A 0.000,B 0.000,C 90.000,E1 38.463} C_DIS
LIN {X 0.170,Y -399.001,Z 766.995,A 0.000,B 0.000,C 90.000,E1 35.105} C_DIS
LIN {X 0.196,Y -399.718,Z 766.976,A 0.000,B 0.000,C 90.000,E1 31.592} C_DIS
LIN {X -0.023,Y -400.868,Z 766.960,A 0.000,B 0.000,C 90.000,E1 28.821} C_DIS
LIN {X -0.065,Y -401.832,Z 766.950,A 0.000,B 0.000,C 90.000,E1 27.078} C_DIS
LIN {X -0.091,Y -402.904,Z 766.941,A 0.000,B 0.000,C 90.000,E1 25.335} C_DIS
LIN {X -0.163,Y -403.811,Z 766.933,A 0.000,B 0.000,C 90.000,E1 23.951} C_DIS
LIN {X -0.130,Y -405.164,Z 766.923,A 0.000,B 0.000,C 90.000,E1 22.206} C_DIS
LIN {X 0.078,Y -408.982,Z 766.902,A 0.000,B 0.000,C 90.000,E1 18.362} C_DIS
LIN {X 0.067,Y -412.679,Z 766.887,A 0.000,B 0.000,C 90.000,E1 15.607} C_DIS
LIN {X -0.095,Y -416.262,Z 766.873,A 0.000,B 0.000,C 90.000,E1 13.231} C_DIS
LIN {X -0.098,Y -419.564,Z 766.862,A 0.000,B 0.000,C 90.000,E1 11.186} C_DIS
LIN {X -0.167,Y -422.362,Z 766.853,A 0.000,B 0.000,C 90.000,E1 9.500} C_DIS
LIN {X -0.098,Y -425.816,Z 766.841,A 0.000,B 0.000,C 90.000,E1 7.466} C_DIS
LIN {X -0.011,Y -429.809,Z 766.828,A 0.000,B 0.000,C 90.000,E1 5.106} C_DIS
LIN {X 0.158,Y -434.058,Z 766.815,A 0.000,B 0.000,C 90.000,E1 2.751} C_DIS
LIN {X 0.202,Y -437.206,Z 766.806,A 0.000,B 0.000,C 90.000,E1 1.088} C_DIS
LIN {X -0.044,Y -441.158,Z 766.795,A 0.000,B 0.000,C 90.000,E1 359.141} C_DIS
LIN {X 0.118,Y -446.667,Z 766.781,A 0.000,B 0.000,C 90.000,E1 356.502} C_DIS
LIN {X -0.119,Y -451.904,Z 766.768,A 0.000,B 0.000,C 90.000,E1 354.261} C_DIS
LIN {X -0.106,Y -455.679,Z 766.759,A 0.000,B 0.000,C 90.000,E1 352.648} C_DIS
LIN {X -0.192,Y -458.580,Z 766.752,A 0.000,B 0.000,C 90.000,E1 351.376} C_DIS
LIN {X -0.161,Y -461.370,Z 766.745,A 0.000,B 0.000,C 90.000,E1 350.095} C_DIS
LIN {X -0.084,Y -464.016,Z 766.738,A 0.000,B 0.000,C 90.000,E1 348.814} C_DIS
LIN {X 0.199,Y -467.908,Z 766.727,A 0.000,B 0.000,C 90.000,E1 346.881} C_DIS
LIN {X 0.200,Y -470.107,Z 766.722,A 0.000,B 0.000,C 90.000,E1 345.936} C_DIS
LIN {X -0.050,Y -472.087,Z 766.719,A 0.000,B 0.000,C 90.000,E1 345.338} C_DIS
LIN {X 0.227,Y -473.292,Z 766.717,A 0.000,B 0.000,C 90.000,E1 344.991} C_DIS
LIN {X -0.201,Y -475.758,Z 766.714,A 0.000,B 0.000,C 90.000,E1 344.574} C_DIS
LIN {X -0.161,Y -478.840,Z 766.712,A 0.000,B 0.000,C 90.000,E1 344.102} C_DIS
LIN {X -0.196,Y -481.883,Z 766.710,A 0.000,B 0.000,C 90.000,E1 343.740} C_DIS
LIN {X 0.197,Y -486.979,Z 766.707,A 0.000,B 0.000,C 90.000,E1 343.196} C_DIS
LIN {X 0.032,Y -492.450,Z 766.704,A 0.000,B 0.000,C 90.000,E1 342.779} C_DIS
LIN {X 0.201,Y -508.293,Z 766.698,A 0.000,B 0.000,C 90.000,E1 341.638} C_DIS
LIN {X -0.184,Y -533.700,Z 766.689,A 0.000,B 0.000,C 90.000,E1 340.061} C_DIS
LIN {X -0.036,Y -538.405,Z 766.688,A 0.000,B 0.000,C 90.000,E1 339.752} C_DIS
LIN {X -0.031,Y -547.498,Z 766.684,A 0.000,B 0.000,C 90.000,E1 339.135} C_DIS
LIN {X -0.313,Y -553.080,Z 766.682,A 0.000,B 0.000,C 90.000,E1 338.720} C_DIS
LIN {X -0.142,Y -559.777,Z 766.678,A 0.000,B 0.000,C 90.000,E1 338.103} C_DIS
LIN {X -0.164,Y -564.920,Z 766.675,A 0.000,B 0.000,C 90.000,E1 337.592} C_DIS
LIN {X 0.027,Y -571.000,Z 766.672,A 0.000,B 0.000,C 90.000,E1 336.922} C_DIS
LIN {X 0.229,Y -575.699,Z 766.669,A 0.000,B 0.000,C 90.000,E1 336.357} C_DIS
LIN {X -0.080,Y -580.171,Z 766.666,A 0.000,B 0.000,C 90.000,E1 335.845} C_DIS
LIN {X -0.207,Y -587.452,Z 766.661,A 0.000,B 0.000,C 90.000,E1 334.921} C_DIS
LIN {X -0.012,Y -593.349,Z 766.656,A 0.000,B 0.000,C 90.000,E1 334.101} C_DIS
LIN {X -0.064,Y -599.874,Z 766.651,A 0.000,B 0.000,C 90.000,E1 333.179} C_DIS
LIN {X 0.262,Y -605.293,Z 766.647,A 0.000,B 0.000,C 90.000,E1 332.359} C_DIS
LIN {X 0.351,Y -612.076,Z 766.641,A 0.000,B 0.000,C 90.000,E1 331.307} C_DIS
LIN {X -0.305,Y -618.444,Z 766.635,A 0.000,B 0.000,C 90.000,E1 330.333} C_DIS
LIN {X -0.036,Y -623.158,Z 766.631,A 0.000,B 0.000,C 90.000,E1 329.537} C_DIS
LIN {X -0.249,Y -628.270,Z 766.626,A 0.000,B 0.000,C 90.000,E1 328.663} C_DIS
LIN {X 0.130,Y -633.165,Z 766.621,A 0.000,B 0.000,C 90.000,E1 327.740} C_DIS
LIN {X 0.010,Y -637.121,Z 766.617,A 0.000,B 0.000,C 90.000,E1 326.993} C_DIS
LIN {X 0.282,Y -640.801,Z 766.612,A 0.000,B 0.000,C 90.000,E1 326.215} C_DIS
LIN {X -0.253,Y -645.444,Z 766.607,A 0.000,B 0.000,C 90.000,E1 325.261} C_DIS
LIN {X 0.106,Y -648.702,Z 766.603,A 0.000,B 0.000,C 90.000,E1 324.482} C_DIS
LIN {X 0.036,Y -652.910,Z 766.597,A 0.000,B 0.000,C 90.000,E1 323.497} C_DIS
LIN {X -0.048,Y -655.854,Z 766.593,A 0.000,B 0.000,C 90.000,E1 322.763} C_DIS
LIN {X -0.080,Y -660.468,Z 766.586,A 0.000,B 0.000,C 90.000,E1 321.537} C_DIS
LIN {X -0.069,Y -665.494,Z 766.578,A 0.000,B 0.000,C 90.000,E1 320.070} C_DIS
LIN {X -0.041,Y -669.416,Z 766.571,A 0.000,B 0.000,C 90.000,E1 318.852} C_DIS
LIN {X 0.038,Y -672.312,Z 766.566,A 0.000,B 0.000,C 90.000,E1 317.877} C_DIS
LIN {X 0.110,Y -674.940,Z 766.561,A 0.000,B 0.000,C 90.000,E1 316.905} C_DIS
LIN {X -0.241,Y -677.380,Z 766.555,A 0.000,B 0.000,C 90.000,E1 315.972} C_DIS
LIN {X -0.093,Y -679.578,Z 766.550,A 0.000,B 0.000,C 90.000,E1 315.000} C_DIS
LIN {X 0.131,Y -682.058,Z 766.543,A 0.000,B 0.000,C 90.000,E1 313.785} C_DIS
LIN {X -0.079,Y -684.387,Z 766.537,A 0.000,B 0.000,C 90.000,E1 312.609} C_DIS
LIN {X -0.316,Y -686.062,Z 766.531,A 0.000,B 0.000,C 90.000,E1 311.676} C_DIS
LIN {X 0.044,Y -687.943,Z 766.525,A 0.000,B 0.000,C 90.000,E1 310.458} C_DIS
LIN {X -0.071,Y -689.160,Z 766.520,A 0.000,B 0.000,C 90.000,E1 309.519} C_DIS
LIN {X -0.039,Y -690.860,Z 766.512,A 0.000,B 0.000,C 90.000,E1 308.096} C_DIS
LIN {X -0.109,Y -691.850,Z 766.506,A 0.000,B 0.000,C 90.000,E1 307.156} C_DIS
LIN {X 0.033,Y -692.953,Z 766.500,A 0.000,B 0.000,C 90.000,E1 305.964} C_DIS
LIN {X 0.243,Y -694.122,Z 766.492,A 0.000,B 0.000,C 90.000,E1 304.532} C_DIS
LIN {X -0.320,Y -695.182,Z 766.484,A 0.000,B 0.000,C 90.000,E1 303.166} C_DIS
LIN {X 0.341,Y -696.446,Z 766.475,A 0.000,B 0.000,C 90.000,E1 301.465} C_DIS
LIN {X 0.148,Y -697.121,Z 766.470,A 0.000,B 0.000,C 90.000,E1 300.541} C_DIS
LIN {X -0.034,Y -697.601,Z 766.465,A 0.000,B 0.000,C 90.000,E1 299.617} C_DIS
LIN {X -0.297,Y -698.149,Z 766.457,A 0.000,B 0.000,C 90.000,E1 298.231} C_DIS
LIN {X 0.003,Y -698.831,Z 766.448,A 0.000,B 0.000,C 90.000,E1 296.565} C_DIS
LIN {X 0.051,Y -699.581,Z 766.440,A 0.000,B 0.000,C 90.000,E1 295.155} C_DIS
LIN {X -0.047,Y -699.763,Z 766.437,A 0.000,B 0.000,C 90.000,E1 294.695} C_DIS
LIN {X 0.199,Y -699.423,Z 766.435,A 0.000,B 0.000,C 90.000,E1 294.207} C_DIS
LIN {X -0.174,Y -699.071,Z 766.433,A 0.000,B 0.000,C 90.000,E1 294.003} C_DIS
LIN {X 0.073,Y -697.463,Z 766.431,A 0.000,B 0.000,C 90.000,E1 293.515} C_DIS
LIN {X 0.331,Y -696.264,Z 766.429,A 0.000,B 0.000,C 90.000,E1 293.259} C_DIS
LIN {X 0.185,Y -695.179,Z 766.429,A 0.000,B 0.000,C 90.000,E1 293.153} C_DIS
LIN {X 0.148,Y -691.103,Z 766.427,A 0.000,B 0.000,C 90.000,E1 292.823} C_DIS
LIN {X 0.151,Y -689.608,Z 766.426,A 0.000,B 0.000,C 90.000,E1 292.717} C_DIS
LIN {X -0.214,Y -687.747,Z 766.426,A 0.000,B 0.000,C 90.000,E1 292.642} C_DIS
LIN {X -0.117,Y -682.860,Z 766.425,A 0.000,B 0.000,C 90.000,E1 292.461} C_DIS
LIN {X -0.206,Y -674.826,Z 766.424,A 0.000,B 0.000,C 90.000,E1 292.259} C_DIS
LIN {X -0.333,Y -667.434,Z 766.423,A 0.000,B 0.000,C 90.000,E1 292.153} C_DIS
LIN {X -0.152,Y -654.479,Z 766.422,A 0.000,B 0.000,C 90.000,E1 291.972} C_DIS
LIN {X 0.276,Y -644.434,Z 766.421,A 0.000,B 0.000,C 90.000,E1 291.770} C_DIS
LIN {X 0.121,Y -634.872,Z 766.420,A 0.000,B 0.000,C 90.000,E1 291.589} C_DIS
LIN {X -0.226,Y -610.552,Z 766.417,A 0.000,B 0.000,C 90.000,E1 291.046} C_DIS
LIN {X 0.069,Y -593.305,Z 766.414,A 0.000,B 0.000,C 90.000,E1 290.556} C_DIS
LIN {X -0.154,Y -575.741,Z 766.411,A 0.000,B 0.000,C 90.000,E1 290.066} C_DIS
LIN {X -0.119,Y -565.480,Z 766.410,A 0.000,B 0.000,C 90.000,E1 289.758} C_DIS
LIN {X 0.166,Y -558.847,Z 766.408,A 0.000,B 0.000,C 90.000,E1 289.450} C_DIS
LIN {X -0.176,Y -556.561,Z 766.407,A 0.000,B 0.000,C 90.000,E1 289.268} C_DIS
LIN {X -0.214,Y -556.538,Z 766.407,A 0.000,B 0.000,C 90.000,E1 289.268} C_DIS
LIN {X -0.158,Y -555.649,Z 766.406,A 0.000,B 0.000,C 90.000,E1 289.014} C_DIS
LIN {X -0.150,Y -555.244,Z 766.404,A 0.000,B 0.000,C 90.000,E1 288.725} C_DIS
LIN {X -0.026,Y -554.470,Z 766.395,A 0.000,B 0.000,C 90.000,E1 287.040} C_DIS
LIN {X -0.114,Y -553.453,Z 766.381,A 0.000,B 0.000,C 90.000,E1 284.537} C_DIS
LIN {X 0.083,Y -552.951,Z 766.373,A 0.000,B 0.000,C 90.000,E1 283.119} C_DIS
LIN {X -0.272,Y -552.387,Z 766.364,A 0.000,B 0.000,C 90.000,E1 281.478} C_DIS
LIN {X -0.200,Y -551.799,Z 766.354,A 0.000,B 0.000,C 90.000,E1 279.792} C_DIS
LIN {X -0.029,Y -551.153,Z 766.343,A 0.000,B 0.000,C 90.000,E1 277.814} C_DIS
LIN {X -0.182,Y -550.533,Z 766.336,A 0.000,B 0.000,C 90.000,E1 276.429} C_DIS
LIN {X 0.101,Y -549.860,Z 766.329,A 0.000,B 0.000,C 90.000,E1 275.277} C_DIS
LIN {X 0.041,Y -548.451,Z 766.317,A 0.000,B 0.000,C 90.000,E1 273.037} C_DIS
LIN {X -0.160,Y -547.341,Z 766.306,A 0.000,B 0.000,C 90.000,E1 271.088} C_DIS
LIN {X 0.068,Y -546.440,Z 766.298,A 0.000,B 0.000,C 90.000,E1 269.656} C_DIS
LIN {X -0.215,Y -545.295,Z 766.289,A 0.000,B 0.000,C 90.000,E1 267.993} C_DIS
LIN {X 0.050,Y -544.060,Z 766.278,A 0.000,B 0.000,C 90.000,E1 265.988} C_DIS
LIN {X -0.215,Y -542.988,Z 766.268,A 0.000,B 0.000,C 90.000,E1 264.318} C_DIS
LIN {X 0.039,Y -541.706,Z 766.259,A 0.000,B 0.000,C 90.000,E1 262.591} C_DIS
LIN {X -0.143,Y -540.020,Z 766.248,A 0.000,B 0.000,C 90.000,E1 260.622} C_DIS
LIN {X 0.144,Y -539.084,Z 766.242,A 0.000,B 0.000,C 90.000,E1 259.454} C_DIS
LIN {X -0.038,Y -537.916,Z 766.234,A 0.000,B 0.000,C 90.000,E1 258.049} C_DIS
LIN {X 0.002,Y -536.103,Z 766.223,A 0.000,B 0.000,C 90.000,E1 256.047} C_DIS
LIN {X -0.067,Y -534.238,Z 766.213,A 0.000,B 0.000,C 90.000,E1 254.338} C_DIS
LIN {X -0.081,Y -532.561,Z 766.205,A 0.000,B 0.000,C 90.000,E1 252.906} C_DIS
LIN {X 0.034,Y -531.002,Z 766.197,A 0.000,B 0.000,C 90.000,E1 251.456} C_DIS
LIN {X -0.076,Y -529.894,Z 766.192,A 0.000,B 0.000,C 90.000,E1 250.604} C_DIS
LIN {X -0.017,Y -527.902,Z 766.184,A 0.000,B 0.000,C 90.000,E1 249.156} C_DIS
LIN {X -0.111,Y -525.849,Z 766.176,A 0.000,B 0.000,C 90.000,E1 247.720} C_DIS
LIN {X -0.066,Y -523.178,Z 766.167,A 0.000,B 0.000,C 90.000,E1 245.973} C_DIS
LIN {X 0.083,Y -521.342,Z 766.160,A 0.000,B 0.000,C 90.000,E1 244.793} C_DIS
LIN {X 0.089,Y -518.949,Z 766.152,A 0.000,B 0.000,C 90.000,E1 243.332} C_DIS
LIN {X -0.175,Y -516.399,Z 766.144,A 0.000,B 0.000,C 90.000,E1 241.897} C_DIS
LIN {X -0.031,Y -513.528,Z 766.136,A 0.000,B 0.000,C 90.000,E1 240.411} C_DIS
LIN {X -0.139,Y -510.691,Z 766.127,A 0.000,B 0.000,C 90.000,E1 238.948} C_DIS
LIN {X 0.068,Y -508.372,Z 766.121,A 0.000,B 0.000,C 90.000,E1 237.740} C_DIS
LIN {X 0.193,Y -506.623,Z 766.116,A 0.000,B 0.000,C 90.000,E1 236.834} C_DIS
LIN {X 0.021,Y -504.677,Z 766.111,A 0.000,B 0.000,C 90.000,E1 235.960} C_DIS
LIN {X -0.123,Y -501.198,Z 766.103,A 0.000,B 0.000,C 90.000,E1 234.482} C_DIS
LIN {X 0.097,Y -498.268,Z 766.096,A 0.000,B 0.000,C 90.000,E1 233.256} C_DIS
LIN {X 0.019,Y -492.164,Z 766.083,A 0.000,B 0.000,C 90.000,E1 230.848} C_DIS
LIN {X 0.062,Y -486.438,Z 766.069,A 0.000,B 0.000,C 90.000,E1 228.405} C_DIS
LIN {X -0.289,Y -481.770,Z 766.057,A 0.000,B 0.000,C 90.000,E1 226.296} C_DIS
LIN {X -0.091,Y -477.158,Z 766.045,A 0.000,B 0.000,C 90.000,E1 224.109} C_DIS
LIN {X 0.121,Y -473.778,Z 766.036,A 0.000,B 0.000,C 90.000,E1 222.528} C_DIS
LIN {X -0.054,Y -470.348,Z 766.028,A 0.000,B 0.000,C 90.000,E1 220.987} C_DIS
LIN {X -0.005,Y -467.668,Z 766.021,A 0.000,B 0.000,C 90.000,E1 219.725} C_DIS
LIN {X -0.238,Y -464.264,Z 766.012,A 0.000,B 0.000,C 90.000,E1 218.177} C_DIS
LIN {X -0.036,Y -459.621,Z 766.000,A 0.000,B 0.000,C 90.000,E1 215.931} C_DIS
LIN {X 0.140,Y -455.705,Z 765.989,A 0.000,B 0.000,C 90.000,E1 213.992} C_DIS
LIN {X -0.017,Y -451.909,Z 765.978,A 0.000,B 0.000,C 90.000,E1 212.084} C_DIS
LIN {X 0.192,Y -447.601,Z 765.966,A 0.000,B 0.000,C 90.000,E1 209.795} C_DIS
LIN {X 0.163,Y -443.939,Z 765.955,A 0.000,B 0.000,C 90.000,E1 207.847} C_DIS
LIN {X -0.034,Y -441.478,Z 765.948,A 0.000,B 0.000,C 90.000,E1 206.565} C_DIS
LIN {X 0.157,Y -438.460,Z 765.938,A 0.000,B 0.000,C 90.000,E1 204.899} C_DIS
LIN {X 0.151,Y -434.065,Z 765.926,A 0.000,B 0.000,C 90.000,E1 202.589} C_DIS
LIN {X -0.172,Y -430.923,Z 765.916,A 0.000,B 0.000,C 90.000,E1 200.972} C_DIS
LIN {X 0.096,Y -426.497,Z 765.903,A 0.000,B 0.000,C 90.000,E1 198.598} C_DIS
LIN {X 0.129,Y -423.295,Z 765.894,A 0.000,B 0.000,C 90.000,E1 196.913} C_DIS
LIN {X 0.200,Y -418.594,Z 765.881,A 0.000,B 0.000,C 90.000,E1 194.537} C_DIS
LIN {X -0.054,Y -414.235,Z 765.868,A 0.000,B 0.000,C 90.000,E1 192.187} C_DIS
LIN {X -0.101,Y -409.995,Z 765.854,A 0.000,B 0.000,C 90.000,E1 189.792} C_DIS
LIN {X 0.027,Y -407.086,Z 765.845,A 0.000,B 0.000,C 90.000,E1 188.049} C_DIS
LIN {X -0.015,Y -402.458,Z 765.829,A 0.000,B 0.000,C 90.000,E1 185.277} C_DIS
LIN {X 0.138,Y -398.788,Z 765.816,A 0.000,B 0.000,C 90.000,E1 182.808} C_DIS
LIN {X 0.027,Y -394.638,Z 765.798,A 0.000,B 0.000,C 90.000,E1 179.656} C_DIS
LIN {X 0.008,Y -392.213,Z 765.786,A 0.000,B 0.000,C 90.000,E1 177.535} C_DIS
LIN {X 0.181,Y -389.489,Z 765.771,A 0.000,B 0.000,C 90.000,E1 174.666} C_DIS
LIN {X -0.077,Y -387.033,Z 765.753,A 0.000,B 0.000,C 90.000,E1 171.489} C_DIS
LIN {X -0.165,Y -385.438,Z 765.739,A 0.000,B 0.000,C 90.000,E1 168.993} C_DIS
LIN {X -0.081,Y -384.195,Z 765.727,A 0.000,B 0.000,C 90.000,E1 166.825} C_DIS
LIN {X 0.066,Y -383.072,Z 765.713,A 0.000,B 0.000,C 90.000,E1 164.283} C_DIS
LIN {X 0.030,Y -382.061,Z 765.697,A 0.000,B 0.000,C 90.000,E1 161.402} C_DIS
LIN {X -0.011,Y -381.318,Z 765.679,A 0.000,B 0.000,C 90.000,E1 158.156} C_DIS
LIN {X 0.067,Y -381.316,Z 765.665,A 0.000,B 0.000,C 90.000,E1 155.613} C_DIS
LIN {X 0.034,Y -382.142,Z 765.643,A 0.000,B 0.000,C 90.000,E1 151.641} C_DIS
LIN {X -0.029,Y -383.867,Z 765.628,A 0.000,B 0.000,C 90.000,E1 149.125} C_DIS
LIN {X 0.200,Y -386.905,Z 765.612,A 0.000,B 0.000,C 90.000,E1 146.215} C_DIS
LIN {X -0.082,Y -388.357,Z 765.607,A 0.000,B 0.000,C 90.000,E1 145.182} C_DIS
LIN {X -0.056,Y -390.905,Z 765.599,A 0.000,B 0.000,C 90.000,E1 143.749} C_DIS
LIN {X -0.143,Y -392.370,Z 765.595,A 0.000,B 0.000,C 90.000,E1 143.050} C_DIS
LIN {X -0.136,Y -395.396,Z 765.589,A 0.000,B 0.000,C 90.000,E1 141.984} C_DIS
LIN {X 0.134,Y -397.981,Z 765.585,A 0.000,B 0.000,C 90.000,E1 141.251} C_DIS
LIN {X 0.037,Y -400.692,Z 765.582,A 0.000,B 0.000,C 90.000,E1 140.678} C_DIS
LIN {X 0.112,Y -404.291,Z 765.578,A 0.000,B 0.000,C 90.000,E1 140.070} C_DIS
